C09140=1110.762,112.427,-59.197,-179.708,8.252,149.498
C09141=1110.767,112.179,-59.177,-179.709,8.249,149.498
C09142=1110.771,111.930,-59.156,-179.711,8.245,149.498
C09143=1110.776,111.680,-59.137,-179.713,8.242,149.498
C09144=1110.780,111.431,-59.116,-179.714,8.238,149.497
C09145=1110.786,111.182,-59.096,-179.716,8.235,149.497
C09146=1110.791,110.932,-59.077,-179.718,8.231,149.497
C09147=1110.795,110.683,-59.056,-179.720,8.228,149.496
C09148=1110.800,110.434,-59.037,-179.721,8.224,149.496
C09149=1110.805,110.185,-59.016,-179.724,8.221,149.496
C09150=1110.810,109.936,-58.997,-179.726,8.216,149.496
C09151=1110.814,109.687,-58.977,-179.728,8.213,149.495
C09152=1110.819,109.437,-58.957,-179.730,8.209,149.495
C09153=1110.824,109.188,-58.937,-179.732,8.205,149.495
C09154=1110.829,108.940,-58.917,-179.734,8.202,149.494
C09155=1110.834,108.690,-58.898,-179.736,8.198,149.494
C09156=1110.838,108.440,-58.878,-179.738,8.195,149.494
C09157=1110.843,108.192,-58.858,-179.740,8.191,149.494
C09158=1110.848,107.942,-58.838,-179.741,8.187,149.493
C09159=1110.852,107.693,-58.819,-179.743,8.184,149.493
C09160=1110.857,107.444,-58.799,-179.745,8.180,149.493
C09161=1110.861,107.195,-58.779,-179.747,8.176,149.492
C09162=1110.867,106.946,-58.760,-179.749,8.173,149.492
C09163=1110.871,106.697,-58.740,-179.751,8.169,149.492
C09164=1110.876,106.448,-58.720,-179.753,8.165,149.491
C09165=1110.881,106.198,-58.700,-179.754,8.161,149.491
C09166=1110.886,105.949,-58.681,-179.756,8.158,149.491
C09167=1110.890,105.736,-58.664,-179.758,8.154,149.490
C09168=1110.894,105.522,-58.647,-179.759,8.151,149.490
C09169=1110.898,105.308,-58.631,-179.761,8.149,149.490
C09170=1110.902,105.094,-58.613,-179.763,8.145,149.490
C09171=1110.906,104.880,-58.597,-179.764,8.142,149.489
C09172=1110.910,104.666,-58.580,-179.766,8.139,149.489
C09173=1110.914,104.453,-58.563,-179.767,8.135,149.488
C09174=1110.919,104.239,-58.547,-179.769,8.132,149.488
C09175=1110.923,103.989,-58.527,-179.771,8.128,149.488
C09176=1110.928,103.740,-58.507,-179.773,8.125,149.488
C09177=1110.932,103.492,-58.488,-179.774,8.121,149.487
C09178=1110.937,103.242,-58.468,-179.776,8.118,149.487
C09179=1110.942,102.993,-58.448,-179.777,8.114,149.487
C09180=1110.947,102.744,-58.429,-179.779,8.110,149.486
C09181=1110.952,102.494,-58.410,-179.781,8.106,149.486
C09182=1110.957,102.246,-58.391,-179.783,8.103,149.485
C09183=1110.961,101.996,-58.371,-179.784,8.099,149.485
C09184=1110.966,101.747,-58.352,-179.786,8.095,149.485
C09185=1110.971,101.498,-58.332,-179.787,8.091,149.484
C09186=1110.975,101.248,-58.313,-179.789,8.088,149.484
C09187=1110.980,100.999,-58.294,-179.791,8.084,149.483
C09188=1110.985,100.750,-58.274,-179.793,8.080,149.483
C09189=1110.990,100.500,-58.255,-179.794,8.076,149.483
C09190=1110.995,100.252,-58.236,-179.796,8.072,149.482
C09191=1111.000,100.002,-58.216,-179.798,8.069,149.482
C09192=1111.005,99.753,-58.197,-179.800,8.065,149.481
C09193=1111.009,99.504,-58.178,-179.801,8.061,149.481
C09194=1111.014,99.255,-58.158,-179.803,8.057,149.481
C09195=1111.019,99.006,-58.139,-179.804,8.053,149.480
C09196=1111.023,98.756,-58.120,-179.805,8.050,149.480
C09197=1111.029,98.507,-58.101,-179.807,8.046,149.479
C09198=1111.033,98.257,-58.082,-179.808,8.042,149.479
C09199=1111.038,98.009,-58.063,-179.811,8.039,149.479
C09200=1111.043,97.759,-58.043,-179.812,8.035,149.478
C09201=1111.047,97.511,-58.025,-179.814,8.031,149.478
C09202=1111.052,97.261,-58.005,-179.815,8.027,149.477
C09203=1111.058,97.012,-57.986,-179.817,8.023,149.477
C09204=1111.062,96.762,-57.967,-179.819,8.019,149.476
C09205=1111.067,96.514,-57.948,-179.820,8.015,149.476
C09206=1111.071,96.264,-57.929,-179.821,8.012,149.476
C09207=1111.076,96.015,-57.910,-179.823,8.008,149.475
C09208=1111.081,95.765,-57.891,-179.824,8.004,149.475
C09209=1111.086,95.517,-57.872,-179.826,8.001,149.474
C09210=1111.091,95.267,-57.852,-179.827,7.996,149.474
C09211=1111.095,95.019,-57.834,-179.829,7.992,149.473
C09212=1111.100,94.768,-57.815,-179.830,7.988,149.473
C09213=1111.105,94.520,-57.796,-179.831,7.985,149.472
C09214=1111.110,94.270,-57.776,-179.833,7.981,149.472
C09215=1111.115,94.021,-57.758,-179.834,7.978,149.471
C09216=1111.119,93.771,-57.739,-179.836,7.974,149.471
C09217=1111.124,93.523,-57.720,-179.838,7.970,149.471
C09218=1111.129,93.273,-57.701,-179.839,7.966,149.470
C09219=1111.134,93.024,-57.682,-179.840,7.962,149.470
C09220=1111.138,92.775,-57.663,-179.841,7.959,149.469
C09221=1111.143,92.525,-57.645,-179.843,7.955,149.469
C09222=1111.149,92.277,-57.625,-179.845,7.951,149.468
C09223=1111.153,92.062,-57.609,-179.846,7.948,149.468
C09224=1111.156,91.848,-57.593,-179.846,7.945,149.467
C09225=1111.161,91.635,-57.578,-179.847,7.941,149.467
C09226=1111.165,91.421,-57.561,-179.849,7.938,149.467
C09227=1111.169,91.206,-57.545,-179.850,7.934,149.466
C09228=1111.174,90.993,-57.529,-179.851,7.932,149.466
C09229=1111.177,90.779,-57.513,-179.852,7.929,149.465
C09230=1111.181,90.565,-57.497,-179.854,7.925,149.465
C09231=1111.187,90.316,-57.478,-179.855,7.921,149.464
C09232=1111.191,90.066,-57.459,-179.856,7.917,149.464
C09233=1111.195,89.818,-57.440,-179.858,7.913,149.463
C09234=1111.201,89.568,-57.422,-179.859,7.910,149.463
C09235=1111.205,89.319,-57.403,-179.860,7.906,149.462
C09236=1111.211,89.069,-57.384,-179.861,7.902,149.462
C09237=1111.215,88.821,-57.366,-179.863,7.898,149.462
C09238=1111.220,88.571,-57.347,-179.864,7.894,149.461
C09239=1111.225,88.322,-57.328,-179.865,7.891,149.460
C09240=1111.229,88.072,-57.310,-179.867,7.887,149.460
C09241=1111.234,87.824,-57.291,-179.868,7.883,149.459
C09242=1111.240,87.574,-57.272,-179.869,7.880,149.459
C09243=1111.244,87.325,-57.253,-179.870,7.876,149.459
C09244=1111.249,87.076,-57.235,-179.872,7.871,149.458
C09245=1111.254,86.826,-57.217,-179.873,7.868,149.457
C09246=1111.258,86.577,-57.198,-179.874,7.864,149.457
C09247=1111.263,86.328,-57.180,-179.875,7.860,149.456
C09248=1111.269,86.078,-57.161,-179.877,7.856,149.456
C09249=1111.273,85.829,-57.142,-179.877,7.853,149.455
C09250=1111.278,85.580,-57.124,-179.879,7.849,149.455
C09251=1111.283,85.331,-57.106,-179.880,7.846,149.454
C09252=1111.288,85.082,-57.087,-179.881,7.841,149.454
C09253=1111.292,84.832,-57.068,-179.883,7.838,149.453
C09254=1111.297,84.583,-57.050,-179.883,7.834,149.453
C09255=1111.302,84.334,-57.032,-179.885,7.830,149.452
C09256=1111.307,84.084,-57.013,-179.886,7.826,149.452
C09257=1111.312,83.835,-56.995,-179.887,7.823,149.451
C09258=1111.317,83.586,-56.977,-179.888,7.819,149.451
C09259=1111.321,83.337,-56.958,-179.889,7.815,149.450
C09260=1111.326,83.087,-56.940,-179.890,7.812,149.450
C09261=1111.331,82.838,-56.921,-179.892,7.807,149.449
C09262=1111.336,82.589,-56.903,-179.893,7.804,149.449
C09263=1111.341,82.340,-56.885,-179.894,7.800,149.448
C09264=1111.345,82.090,-56.866,-179.895,7.797,149.447
C09265=1111.350,81.841,-56.848,-179.896,7.792,149.447
C09266=1111.356,81.592,-56.830,-179.897,7.789,149.446
C09267=1111.361,81.342,-56.812,-179.898,7.785,149.446
C09268=1111.365,81.092,-56.793,-179.899,7.781,149.445
C09269=1111.369,80.844,-56.775,-179.900,7.778,149.445
C09270=1111.374,80.595,-56.757,-179.902,7.774,149.444
C09271=1111.379,80.346,-56.739,-179.902,7.770,149.444
C09272=1111.384,80.096,-56.721,-179.904,7.766,149.443
C09273=1111.389,79.846,-56.702,-179.904,7.763,149.443
C09274=1111.394,79.597,-56.684,-179.905,7.759,149.442
C09275=1111.399,79.348,-56.666,-179.906,7.756,149.441
C09276=1111.404,79.099,-56.648,-179.907,7.751,149.441
C09277=1111.409,78.849,-56.630,-179.908,7.748,149.440
C09278=1111.413,78.600,-56.611,-179.909,7.744,149.440
C09279=1111.418,78.386,-56.596,-179.910,7.741,149.439
C09280=1111.421,78.172,-56.580,-179.911,7.738,149.439
C09281=1111.426,77.958,-56.565,-179.912,7.734,149.438
C09282=1111.430,77.744,-56.549,-179.913,7.731,149.438
C09283=1111.435,77.530,-56.534,-179.914,7.728,149.437
C09284=1111.438,77.316,-56.518,-179.915,7.725,149.437
C09285=1111.442,77.103,-56.502,-179.916,7.722,149.436
C09286=1111.446,76.888,-56.487,-179.917,7.719,149.436
C09287=1111.451,76.639,-56.469,-179.917,7.715,149.435
C09288=1111.456,76.390,-56.451,-179.919,7.711,149.435
C09289=1111.461,76.141,-56.433,-179.920,7.707,149.435
C09290=1111.466,75.891,-56.415,-179.922,7.703,149.434
C09291=1111.471,75.642,-56.397,-179.923,7.699,149.433
C09292=1111.475,75.392,-56.379,-179.925,7.695,149.433
C09293=1111.480,75.143,-56.361,-179.926,7.691,149.433
C09294=1111.485,74.894,-56.343,-179.927,7.687,149.432
C09295=1111.490,74.645,-56.325,-179.929,7.683,149.431
C09296=1111.495,74.395,-56.307,-179.930,7.679,149.431
C09297=1111.500,74.146,-56.289,-179.932,7.675,149.431
C09298=1111.505,73.897,-56.272,-179.933,7.671,149.430
C09299=1111.510,73.647,-56.254,-179.935,7.667,149.430
C09300=1111.515,73.398,-56.236,-179.936,7.664,149.429
C09301=1111.520,73.149,-56.218,-179.937,7.660,149.428
C09302=1111.524,72.899,-56.199,-179.938,7.656,149.428
C09303=1111.529,72.649,-56.182,-179.940,7.652,149.428
C09304=1111.534,72.400,-56.164,-179.942,7.648,149.427
C09305=1111.539,72.151,-56.146,-179.943,7.644,149.426
C09306=1111.544,71.902,-56.128,-179.944,7.640,149.426
C09307=1111.548,71.653,-56.111,-179.946,7.636,149.426
C09308=1111.553,71.403,-56.093,-179.947,7.632,149.425
C09309=1111.558,71.154,-56.075,-179.948,7.628,149.425
C09310=1111.563,70.905,-56.057,-179.949,7.625,149.424
C09311=1111.568,70.656,-56.039,-179.951,7.620,149.423
C09312=1111.573,70.406,-56.022,-179.952,7.616,149.423
C09313=1111.578,70.157,-56.004,-179.954,7.612,149.423
C09314=1111.582,69.908,-55.987,-179.955,7.608,149.422
C09315=1111.588,69.658,-55.970,-179.956,7.604,149.422
C09316=1111.593,69.409,-55.952,-179.958,7.600,149.421
C09317=1111.597,69.160,-55.934,-179.959,7.596,149.420
C09318=1111.603,68.910,-55.916,-179.961,7.592,149.420
C09319=1111.608,68.661,-55.898,-179.962,7.588,149.420
C09320=1111.612,68.412,-55.881,-179.963,7.585,149.419
C09321=1111.617,68.162,-55.864,-179.964,7.581,149.418
C09322=1111.622,67.913,-55.846,-179.966,7.577,149.418
C09323=1111.627,67.664,-55.828,-179.967,7.573,149.417
C09324=1111.631,67.414,-55.811,-179.969,7.569,149.417
C09325=1111.636,67.165,-55.793,-179.970,7.565,149.417
C09326=1111.641,66.915,-55.776,-179.971,7.561,149.416
C09327=1111.646,66.666,-55.758,-179.973,7.557,149.415
C09328=1111.651,66.417,-55.741,-179.973,7.553,149.415
C09329=1111.656,66.167,-55.723,-179.975,7.549,149.414
C09330=1111.661,65.918,-55.706,-179.976,7.545,149.414
C09331=1111.666,65.669,-55.688,-179.978,7.541,149.413
C09332=1111.670,65.420,-55.671,-179.979,7.537,149.413
C09333=1111.675,65.170,-55.653,-179.981,7.533,149.412
C09334=1111.680,64.921,-55.635,-179.982,7.529,149.412
C09335=1111.684,64.707,-55.621,-179.983,7.526,149.411
C09336=1111.689,64.493,-55.606,-179.984,7.523,149.411
C09337=1111.692,64.279,-55.591,-179.985,7.519,149.410
C09338=1111.697,64.065,-55.576,-179.986,7.516,149.410
C09339=1111.701,63.851,-55.562,-179.987,7.513,149.410
C09340=1111.706,63.637,-55.547,-179.989,7.509,149.409
C09341=1111.710,63.422,-55.531,-179.990,7.506,149.409
C09342=1111.714,63.208,-55.517,-179.991,7.502,149.408
C09343=1111.719,62.959,-55.500,-179.992,7.498,149.408
C09344=1111.723,62.710,-55.482,-179.993,7.494,149.407
C09345=1111.728,62.460,-55.465,-179.994,7.490,149.407
C09346=1111.734,62.210,-55.448,-179.996,7.486,149.406
C09347=1111.738,61.961,-55.430,-179.997,7.483,149.406
C09348=1111.744,61.712,-55.413,-179.998,7.479,149.405
C09349=1111.748,61.463,-55.397,-179.999,7.475,149.405
C09350=1111.753,61.214,-55.379,179.999,7.470,149.404
C09351=1111.757,60.964,-55.362,179.998,7.467,149.404
C09352=1111.763,60.714,-55.345,179.997,7.462,149.403
C09353=1111.768,60.465,-55.327,179.995,7.458,149.402
C09354=1111.773,60.216,-55.310,179.995,7.455,149.402
C09355=1111.778,59.967,-55.293,179.993,7.451,149.401
C09356=1111.782,59.718,-55.276,179.992,7.447,149.401
C09357=1111.787,59.468,-55.259,179.990,7.443,149.400
C09358=1111.792,59.218,-55.242,179.989,7.439,149.400
C09359=1111.797,58.969,-55.225,179.988,7.435,149.399
C09360=1111.802,58.720,-55.208,179.987,7.431,149.399
C09361=1111.807,58.471,-55.190,179.986,7.427,149.398
C09362=1111.811,58.221,-55.174,179.984,7.423,149.398
C09363=1111.817,57.971,-55.156,179.983,7.419,149.397
C09364=1111.821,57.722,-55.140,179.982,7.415,149.397
C09365=1111.827,57.473,-55.123,179.980,7.411,149.396
C09366=1111.831,57.224,-55.105,179.979,7.407,149.396
C09367=1111.836,56.974,-55.088,179.978,7.403,149.395
C09368=1111.841,56.725,-55.072,179.977,7.399,149.394
C09369=1111.847,56.476,-55.055,179.976,7.395,149.394
C09370=1111.851,56.226,-55.038,179.974,7.391,149.393
C09371=1111.856,55.976,-55.021,179.973,7.387,149.393
C09372=1111.861,55.727,-55.004,179.972,7.383,149.392
C09373=1111.866,55.478,-54.988,179.971,7.379,149.392
C09374=1111.871,55.229,-54.970,179.970,7.375,149.391
C09375=1111.875,54.979,-54.953,179.968,7.371,149.391
C09376=1111.881,54.730,-54.936,179.967,7.367,149.390
C09377=1111.886,54.481,-54.920,179.966,7.363,149.389
C09378=1111.890,54.231,-54.903,179.965,7.359,149.389
C09379=1111.895,53.981,-54.886,179.964,7.356,149.388
C09380=1111.900,53.733,-54.869,179.963,7.351,149.388
C09381=1111.906,53.483,-54.852,179.962,7.347,149.387
C09382=1111.910,53.233,-54.835,179.960,7.343,149.387
C09383=1111.915,52.984,-54.819,179.959,7.339,149.386
C09384=1111.920,52.735,-54.802,179.958,7.336,149.386
C09385=1111.925,52.485,-54.785,179.957,7.331,149.385
C09386=1111.929,52.236,-54.768,179.956,7.327,149.384
C09387=1111.935,51.987,-54.752,179.954,7.323,149.384
C09388=1111.940,51.737,-54.735,179.953,7.319,149.383
C09389=1111.944,51.487,-54.719,179.952,7.315,149.383
C09390=1111.950,51.238,-54.702,179.951,7.311,149.382
C09391=1111.954,51.024,-54.688,179.950,7.308,149.382
C09392=1111.959,50.810,-54.674,179.949,7.304,149.381
C09393=1111.962,50.596,-54.659,179.948,7.301,149.381
C09394=1111.967,50.382,-54.644,179.947,7.297,149.380
C09395=1111.971,50.167,-54.630,179.946,7.294,149.380
C09396=1111.975,49.954,-54.616,179.945,7.290,149.379
C09397=1111.979,49.739,-54.602,179.944,7.287,149.379
C09398=1111.983,49.526,-54.588,179.943,7.283,149.378
C09399=1111.989,49.275,-54.571,179.942,7.280,149.378
C09400=1111.993,49.026,-54.555,179.941,7.276,149.377
C09401=1111.998,48.777,-54.538,179.940,7.272,149.376
C09402=1112.003,48.527,-54.522,179.939,7.267,149.376
C09403=1112.009,48.278,-54.505,179.937,7.263,149.375
C09404=1112.013,48.028,-54.489,179.936,7.259,149.375
C09405=1112.018,47.779,-54.472,179.936,7.256,149.374
C09406=1112.023,47.530,-54.456,179.934,7.251,149.373
C09407=1112.027,47.280,-54.439,179.933,7.247,149.373
C09408=1112.034,47.031,-54.423,179.932,7.243,149.372
C09409=1112.038,46.781,-54.406,179.931,7.239,149.372
C09410=1112.043,46.532,-54.390,179.930,7.236,149.371
C09411=1112.048,46.283,-54.373,179.929,7.231,149.371
C09412=1112.052,46.033,-54.357,179.928,7.227,149.370
C09413=1112.057,45.784,-54.341,179.927,7.223,149.369
C09414=1112.062,45.535,-54.324,179.925,7.219,149.369
C09415=1112.068,45.285,-54.308,179.925,7.215,149.368
C09416=1112.073,45.035,-54.292,179.923,7.211,149.368
C09417=1112.078,44.787,-54.275,179.922,7.207,149.367
C09418=1112.082,44.537,-54.259,179.921,7.203,149.366
C09419=1112.087,44.287,-54.243,179.920,7.198,149.366
C09420=1112.092,44.038,-54.226,179.919,7.194,149.365
C09421=1112.097,43.788,-54.210,179.918,7.191,149.364
C09422=1112.102,43.539,-54.194,179.917,7.187,149.364
C09423=1112.107,43.289,-54.178,179.916,7.182,149.363
C09424=1112.112,43.040,-54.162,179.915,7.178,149.363
C09425=1112.117,42.791,-54.145,179.913,7.174,149.362
C09426=1112.122,42.541,-54.129,179.913,7.170,149.361
C09427=1112.127,42.292,-54.112,179.911,7.166,149.361
C09428=1112.132,42.042,-54.097,179.910,7.162,149.360
C09429=1112.137,41.793,-54.080,179.909,7.158,149.360
C09430=1112.142,41.544,-54.064,179.908,7.154,149.359
C09431=1112.147,41.294,-54.048,179.908,7.150,149.358
C09432=1112.152,41.045,-54.032,179.907,7.146,149.358
C09433=1112.156,40.795,-54.015,179.905,7.142,149.357
C09434=1112.162,40.546,-54.000,179.904,7.137,149.357
C09435=1112.167,40.297,-53.984,179.903,7.133,149.356
C09436=1112.172,40.047,-53.968,179.903,7.130,149.355
C09437=1112.177,39.798,-53.951,179.901,7.125,149.355
C09438=1112.182,39.548,-53.935,179.900,7.121,149.354
C09439=1112.187,39.299,-53.920,179.899,7.117,149.353
C09440=1112.191,39.049,-53.903,179.898,7.112,149.353
C09441=1112.197,38.800,-53.888,179.897,7.108,149.352
C09442=1112.201,38.550,-53.871,179.896,7.105,149.352
C09443=1112.207,38.301,-53.855,179.895,7.101,149.351
C09444=1112.211,38.052,-53.840,179.894,7.096,149.350
C09445=1112.216,37.802,-53.824,179.893,7.092,149.350
C09446=1112.221,37.553,-53.808,179.892,7.088,149.349
C09447=1112.225,37.338,-53.794,179.892,7.084,149.348
C09448=1112.230,37.124,-53.781,179.891,7.081,149.348
C09449=1112.234,36.910,-53.767,179.890,7.078,149.347
C09450=1112.238,36.696,-53.753,179.889,7.074,149.347
C09451=1112.243,36.481,-53.740,179.888,7.070,149.346
C09452=1112.247,36.267,-53.726,179.887,7.067,149.346
C09453=1112.251,36.053,-53.712,179.887,7.064,149.345
C09454=1112.256,35.838,-53.698,179.886,7.059,149.344
C09455=1112.261,35.589,-53.682,179.885,7.055,149.344
C09456=1112.266,35.340,-53.666,179.884,7.051,149.343
C09457=1112.270,35.090,-53.651,179.883,7.047,149.342
C09458=1112.275,34.841,-53.636,179.882,7.043,149.342
C09459=1112.280,34.591,-53.619,179.881,7.038,149.341
C09460=1112.285,34.342,-53.603,179.880,7.034,149.341
C09461=1112.291,34.093,-53.588,179.880,7.031,149.340
C09462=1112.295,33.842,-53.572,179.878,7.026,149.339
C09463=1112.300,33.594,-53.556,179.877,7.022,149.339
C09464=1112.305,33.345,-53.540,179.876,7.018,149.338
C09465=1112.310,33.094,-53.524,179.875,7.013,149.337
C09466=1112.315,32.845,-53.509,179.875,7.010,149.337
C09467=1112.321,32.596,-53.493,179.874,7.006,149.336
C09468=1112.325,32.346,-53.478,179.873,7.001,149.335
C09469=1112.330,32.097,-53.462,179.872,6.997,149.335
C09470=1112.335,31.848,-53.446,179.871,6.993,149.334
C09471=1112.341,31.598,-53.430,179.870,6.989,149.333
C09472=1112.345,31.348,-53.415,179.869,6.985,149.333
C09473=1112.350,31.099,-53.400,179.868,6.980,149.332
C09474=1112.355,30.850,-53.384,179.867,6.976,149.331
C09475=1112.360,30.600,-53.368,179.866,6.971,149.330
C09476=1112.365,30.350,-53.353,179.865,6.967,149.330
C09477=1112.370,30.101,-53.337,179.865,6.964,149.329
C09478=1112.376,29.852,-53.322,179.864,6.959,149.329
C09479=1112.379,29.603,-53.306,179.863,6.955,149.328
C09480=1112.385,29.353,-53.290,179.862,6.951,149.327
C09481=1112.390,29.104,-53.275,179.861,6.946,149.326
C09482=1112.394,28.854,-53.259,179.861,6.942,149.326
C09483=1112.400,28.605,-53.244,179.860,6.938,149.325
C09484=1112.405,28.355,-53.228,179.859,6.934,149.324
C09485=1112.410,28.106,-53.213,179.858,6.930,149.324
C09486=1112.415,27.857,-53.197,179.857,6.925,149.323
C09487=1112.420,27.607,-53.182,179.856,6.921,149.322
C09488=1112.424,27.357,-53.167,179.855,6.917,149.322
C09489=1112.430,27.107,-53.152,179.854,6.913,149.321
C09490=1112.436,26.858,-53.136,179.854,6.908,149.320
C09491=1112.440,26.608,-53.121,179.853,6.904,149.319
C09492=1112.445,26.359,-53.105,179.852,6.899,149.319
C09493=1112.450,26.110,-53.090,179.851,6.896,149.318
C09494=1112.455,25.860,-53.075,179.851,6.891,149.317
C09495=1112.460,25.611,-53.059,179.850,6.887,149.316
C09496=1112.464,25.361,-53.044,179.849,6.883,149.316
C09497=1112.470,25.112,-53.028,179.848,6.878,149.315
C09498=1112.475,24.863,-53.013,179.847,6.874,149.314
C09499=1112.480,24.613,-52.998,179.847,6.870,149.314
C09500=1112.486,24.363,-52.983,179.845,6.866,149.313
C09501=1112.490,24.114,-52.968,179.845,6.861,149.312
C09502=1112.495,23.864,-52.952,179.844,6.857,149.311
C09503=1112.499,23.650,-52.940,179.843,6.853,149.311
C09504=1112.504,23.436,-52.926,179.843,6.850,149.310
C09505=1112.508,23.221,-52.912,179.842,6.845,149.309
C09506=1112.512,23.007,-52.900,179.842,6.842,149.309
C09507=1112.516,22.792,-52.886,179.841,6.839,149.308
C09508=1112.521,22.579,-52.874,179.840,6.834,149.308
C09509=1112.525,22.364,-52.860,179.839,6.831,149.307
C09510=1112.530,22.149,-52.847,179.839,6.827,149.306
C09511=1112.534,21.900,-52.832,179.838,6.823,149.306
C09512=1112.540,21.651,-52.817,179.837,6.818,149.305
C09513=1112.545,21.401,-52.802,179.836,6.814,149.304
C09514=1112.550,21.152,-52.787,179.836,6.810,149.303
C09515=1112.555,20.903,-52.772,179.835,6.806,149.303
C09516=1112.559,20.652,-52.756,179.834,6.801,149.302
C09517=1112.564,20.403,-52.742,179.833,6.797,149.301
C09518=1112.569,20.154,-52.727,179.833,6.792,149.300
C09519=1112.574,19.904,-52.711,179.832,6.788,149.300
C09520=1112.579,19.655,-52.697,179.831,6.783,149.299
C09521=1112.585,19.405,-52.681,179.831,6.779,149.298
C09522=1112.589,19.156,-52.666,179.830,6.775,149.297
C09523=1112.595,18.906,-52.651,179.829,6.770,149.297
C09524=1112.600,18.657,-52.636,179.829,6.766,149.296
C09525=1112.605,18.407,-52.622,179.828,6.761,149.295
C09526=1112.610,18.158,-52.606,179.827,6.757,149.294
C09527=1112.615,17.909,-52.591,179.827,6.753,149.293
C09528=1112.620,17.659,-52.577,179.826,6.748,149.293
C09529=1112.625,17.410,-52.562,179.825,6.744,149.292
C09530=1112.629,17.159,-52.547,179.824,6.739,149.291
C09531=1112.635,16.910,-52.531,179.823,6.735,149.290
C09532=1112.640,16.660,-52.517,179.823,6.730,149.290
C09533=1112.644,16.411,-52.502,179.822,6.726,149.289
C09534=1112.650,16.162,-52.487,179.822,6.722,149.288
C09535=1112.655,15.912,-52.472,179.821,6.717,149.287
C09536=1112.659,15.663,-52.457,179.820,6.713,149.286
C09537=1112.665,15.413,-52.442,179.820,6.708,149.286
C09538=1112.670,15.164,-52.427,179.819,6.704,149.285
C09539=1112.675,14.914,-52.413,179.818,6.699,149.284
C09540=1112.680,14.665,-52.398,179.818,6.695,149.283
C09541=1112.685,14.415,-52.383,179.818,6.691,149.282
C09542=1112.690,14.165,-52.369,179.817,6.686,149.282
C09543=1112.695,13.916,-52.354,179.816,6.682,149.281
C09544=1112.700,13.666,-52.339,179.815,6.677,149.280
C09545=1112.705,13.417,-52.324,179.814,6.673,149.279
C09546=1112.710,13.167,-52.310,179.814,6.668,149.278
C09547=1112.715,12.918,-52.295,179.813,6.663,149.277
C09548=1112.720,12.668,-52.280,179.813,6.660,149.277
C09549=1112.725,12.418,-52.266,179.812,6.655,149.276
C09550=1112.730,12.169,-52.251,179.812,6.650,149.275
C09551=1112.735,11.920,-52.237,179.811,6.646,149.274
C09552=1112.741,11.670,-52.222,179.810,6.641,149.273
C09553=1112.746,11.421,-52.207,179.810,6.637,149.273
C09554=1112.751,11.171,-52.193,179.809,6.632,149.272
C09555=1112.755,10.922,-52.178,179.809,6.627,149.271
C09556=1112.760,10.673,-52.163,179.809,6.623,149.270
C09557=1112.766,10.423,-52.149,179.808,6.619,149.269
C09558=1112.771,10.173,-52.134,179.807,6.614,149.268
C09559=1112.775,9.959,-52.121,179.806,6.610,149.268
C09560=1112.780,9.745,-52.108,179.806,6.606,149.267
C09561=1112.784,9.530,-52.096,179.806,6.603,149.266
C09562=1112.788,9.316,-52.084,179.805,6.598,149.265
C09563=1112.793,9.101,-52.071,179.805,6.594,149.265
C09564=1112.797,8.887,-52.059,179.804,6.591,149.264
C09565=1112.801,8.673,-52.047,179.803,6.586,149.263
C09566=1112.806,8.458,-52.034,179.803,6.582,149.262
C09567=1112.811,8.208,-52.019,179.803,6.578,149.261
C09568=1112.816,7.958,-52.005,179.802,6.573,149.261
C09569=1112.821,7.710,-51.990,179.801,6.569,149.260
C09570=1112.826,7.460,-51.976,179.801,6.564,149.259
C09571=1112.831,7.210,-51.962,179.800,6.559,149.258
C09572=1112.836,6.961,-51.948,179.800,6.555,149.257
C09573=1112.841,6.711,-51.933,179.800,6.551,149.256
C09574=1112.846,6.461,-51.919,179.799,6.546,149.256
C09575=1112.850,6.212,-51.904,179.798,6.542,149.255
C09576=1112.856,5.962,-51.889,179.798,6.537,149.254
C09577=1112.861,5.713,-51.875,179.797,6.532,149.253
C09578=1112.866,5.463,-51.861,179.796,6.528,149.252
C09579=1112.871,5.214,-51.847,179.795,6.523,149.252
C09580=1112.876,4.964,-51.832,179.795,6.518,149.251
C09581=1112.881,4.714,-51.818,179.794,6.514,149.250
C09582=1112.886,4.465,-51.804,179.794,6.509,149.249
C09583=1112.892,4.216,-51.790,179.793,6.505,149.248
C09584=1112.896,3.967,-51.775,179.792,6.500,149.247
C09585=1112.901,3.717,-51.761,179.792,6.496,149.246
C09586=1112.906,3.467,-51.746,179.792,6.491,149.246
C09587=1112.911,3.217,-51.732,179.791,6.487,149.245
C09588=1112.917,2.968,-51.718,179.790,6.482,149.244
C09589=1112.922,2.719,-51.704,179.790,6.478,149.243
C09590=1112.927,2.469,-51.690,179.789,6.473,149.242
C09591=1112.932,2.219,-51.675,179.789,6.468,149.241
C09592=1112.937,1.970,-51.662,179.788,6.464,149.241
C09593=1112.942,1.721,-51.647,179.787,6.459,149.240
C09594=1112.947,1.471,-51.633,179.787,6.454,149.239
C09595=1112.952,1.221,-51.619,179.787,6.451,149.238
C09596=1112.957,0.971,-51.604,179.786,6.446,149.237
C09597=1112.962,0.723,-51.591,179.785,6.441,149.236
C09598=1112.967,0.473,-51.577,179.785,6.437,149.236
C09599=1112.972,0.223,-51.563,179.784,6.432,149.235
C09600=1112.977,-0.027,-51.549,179.783,6.428,149.234
C09601=1112.983,-0.276,-51.535,179.783,6.423,149.233
C09602=1112.988,-0.526,-51.521,179.782,6.418,149.232
C09603=1112.993,-0.775,-51.507,179.781,6.414,149.232
C09604=1112.998,-1.024,-51.493,179.781,6.409,149.231
C09605=1113.003,-1.274,-51.478,179.781,6.405,149.230
C09606=1113.008,-1.524,-51.464,179.780,6.401,149.229
C09607=1113.012,-1.773,-51.450,179.779,6.396,149.228
C09608=1113.018,-2.023,-51.437,179.779,6.392,149.227
C09609=1113.023,-2.273,-51.423,179.778,6.387,149.226
C09610=1113.028,-2.522,-51.409,179.777,6.382,149.226
C09611=1113.034,-2.771,-51.395,179.777,6.378,149.225
C09612=1113.038,-3.021,-51.380,179.776,6.373,149.224
C09613=1113.044,-3.271,-51.367,179.775,6.369,149.223
C09614=1113.049,-3.520,-51.354,179.775,6.365,149.222
C09615=1113.052,-3.735,-51.341,179.774,6.360,149.222
C09616=1113.057,-3.949,-51.330,179.774,6.357,149.221
C09617=1113.061,-4.164,-51.317,179.773,6.352,149.220
C09618=1113.066,-4.378,-51.305,179.773,6.349,149.220
C09619=1113.070,-4.593,-51.293,179.772,6.345,149.219
C09620=1113.075,-4.807,-51.281,179.771,6.341,149.218
C09621=1113.080,-5.022,-51.270,179.771,6.337,149.218
C09622=1113.084,-5.237,-51.257,179.771,6.333,149.217
C09623=1113.088,-5.486,-51.244,179.770,6.329,149.216
C09624=1113.094,-5.736,-51.231,179.770,6.324,149.215
C09625=1113.099,-5.985,-51.216,179.769,6.320,149.214
C09626=1113.104,-6.234,-51.202,179.768,6.315,149.214
C09627=1113.109,-6.484,-51.189,179.768,6.310,149.213
C09628=1113.114,-6.734,-51.175,179.767,6.306,149.212
C09629=1113.119,-6.983,-51.161,179.767,6.301,149.211
C09630=1113.124,-7.233,-51.148,179.766,6.298,149.210
C09631=1113.129,-7.483,-51.134,179.766,6.293,149.209
C09632=1113.134,-7.732,-51.121,179.765,6.288,149.208
C09633=1113.139,-7.982,-51.106,179.764,6.284,149.208
C09634=1113.144,-8.231,-51.093,179.764,6.279,149.207
C09635=1113.150,-8.481,-51.080,179.763,6.274,149.206
C09636=1113.155,-8.730,-51.066,179.763,6.270,149.205
C09637=1113.160,-8.980,-51.053,179.762,6.265,149.204
C09638=1113.165,-9.230,-51.038,179.761,6.261,149.204
C09639=1113.170,-9.479,-51.025,179.761,6.256,149.203
C09640=1113.175,-9.729,-51.012,179.760,6.252,149.202
C09641=1113.180,-9.978,-50.998,179.760,6.248,149.201
C09642=1113.185,-10.228,-50.984,179.759,6.243,149.200
C09643=1113.190,-10.478,-50.970,179.759,6.238,149.199
C09644=1113.196,-10.727,-50.957,179.758,6.234,149.199
C09645=1113.200,-10.977,-50.943,179.757,6.229,149.198
C09646=1113.206,-11.226,-50.930,179.757,6.224,149.197
C09647=1113.211,-11.476,-50.916,179.756,6.220,149.196
C09648=1113.216,-11.725,-50.903,179.755,6.215,149.195
C09649=1113.221,-11.975,-50.889,179.755,6.211,149.194
C09650=1113.227,-12.225,-50.876,179.754,6.206,149.194
C09651=1113.231,-12.474,-50.862,179.754,6.201,149.193
C09652=1113.237,-12.724,-50.849,179.753,6.198,149.192
C09653=1113.241,-12.973,-50.835,179.753,6.193,149.191
C09654=1113.247,-13.223,-50.822,179.752,6.188,149.190
C09655=1113.251,-13.473,-50.809,179.752,6.183,149.189
C09656=1113.257,-13.722,-50.795,179.751,6.179,149.189
C09657=1113.261,-13.972,-50.782,179.750,6.174,149.188
C09658=1113.267,-14.221,-50.768,179.750,6.170,149.187
C09659=1113.272,-14.471,-50.755,179.749,6.165,149.186
C09660=1113.277,-14.720,-50.742,179.749,6.160,149.185
C09661=1113.282,-14.970,-50.728,179.748,6.156,149.184
C09662=1113.287,-15.219,-50.715,179.747,6.151,149.183
C09663=1113.293,-15.470,-50.702,179.747,6.146,149.183
C09664=1113.297,-15.718,-50.689,179.746,6.142,149.182
C09665=1113.303,-15.969,-50.675,179.746,6.137,149.181
C09666=1113.308,-16.218,-50.662,179.745,6.133,149.180
C09667=1113.312,-16.468,-50.649,179.745,6.129,149.179
C09668=1113.318,-16.717,-50.635,179.745,6.124,149.178
C09669=1113.323,-16.966,-50.623,179.744,6.119,149.177
C09670=1113.328,-17.217,-50.609,179.744,6.114,149.177
C09671=1113.333,-17.431,-50.598,179.743,6.110,149.176
C09672=1113.337,-17.645,-50.587,179.742,6.107,149.175
C09673=1113.341,-17.860,-50.575,179.742,6.102,149.174
C09674=1113.346,-18.075,-50.564,179.741,6.098,149.174
C09675=1113.350,-18.289,-50.552,179.741,6.095,149.173
C09676=1113.354,-18.504,-50.542,179.741,6.090,149.172
C09677=1113.359,-18.719,-50.530,179.740,6.086,149.171
C09678=1113.363,-18.933,-50.519,179.739,6.082,149.171
C09679=1113.369,-19.183,-50.506,179.739,6.077,149.170
C09680=1113.374,-19.433,-50.492,179.738,6.073,149.169
C09681=1113.379,-19.682,-50.479,179.738,6.068,149.168
C09682=1113.383,-19.932,-50.466,179.737,6.063,149.167
C09683=1113.389,-20.181,-50.453,179.737,6.058,149.166
C09684=1113.394,-20.431,-50.440,179.736,6.054,149.165
C09685=1113.399,-20.681,-50.427,179.736,6.049,149.164
C09686=1113.404,-20.930,-50.414,179.735,6.044,149.164
C09687=1113.410,-21.180,-50.402,179.735,6.040,149.163
C09688=1113.415,-21.429,-50.387,179.734,6.035,149.162
C09689=1113.420,-21.679,-50.375,179.734,6.030,149.161
C09690=1113.425,-21.928,-50.362,179.733,6.026,149.160
C09691=1113.430,-22.178,-50.349,179.732,6.021,149.159
C09692=1113.435,-22.428,-50.336,179.732,6.016,149.158
C09693=1113.440,-22.677,-50.323,179.731,6.012,149.157
C09694=1113.446,-22.927,-50.310,179.731,6.007,149.157
C09695=1113.451,-23.177,-50.297,179.731,6.002,149.156
C09696=1113.456,-23.426,-50.285,179.730,5.997,149.155
C09697=1113.461,-23.676,-50.271,179.730,5.993,149.154
C09698=1113.466,-23.926,-50.258,179.729,5.988,149.153
C09699=1113.471,-24.175,-50.246,179.729,5.983,149.152
C09700=1113.476,-24.425,-50.233,179.729,5.978,149.151
C09701=1113.482,-24.675,-50.220,179.728,5.973,149.150
C09702=1113.487,-24.924,-50.207,179.728,5.969,149.149
C09703=1113.492,-25.173,-50.194,179.727,5.964,149.148
C09704=1113.496,-25.423,-50.181,179.727,5.959,149.147
C09705=1113.502,-25.673,-50.168,179.726,5.954,149.146
C09706=1113.507,-25.922,-50.156,179.726,5.950,149.146
C09707=1113.512,-26.172,-50.143,179.726,5.945,149.144
C09708=1113.517,-26.422,-50.130,179.727,5.941,149.143
C09709=1113.522,-26.671,-50.117,179.727,5.937,149.142
C09710=1113.528,-26.920,-50.104,179.728,5.933,149.141
C09711=1113.533,-27.171,-50.092,179.727,5.928,149.140
C09712=1113.538,-27.420,-50.079,179.728,5.924,149.139
C09713=1113.543,-27.670,-50.067,179.728,5.920,149.138
C09714=1113.548,-27.919,-50.054,179.728,5.916,149.137
C09715=1113.554,-28.169,-50.041,179.728,5.911,149.136
C09716=1113.559,-28.419,-50.028,179.728,5.907,149.135
C09717=1113.564,-28.668,-50.015,179.728,5.903,149.134
C09718=1113.569,-28.917,-50.003,179.729,5.898,149.133
C09719=1113.574,-29.168,-49.991,179.729,5.894,149.132
C09720=1113.579,-29.417,-49.978,179.728,5.889,149.131
C09721=1113.584,-29.667,-49.965,179.728,5.885,149.131
C09722=1113.590,-29.916,-49.952,179.728,5.881,149.130
C09723=1113.594,-30.166,-49.939,179.728,5.876,149.129
C09724=1113.600,-30.416,-49.927,179.729,5.872,149.128
C09725=1113.605,-30.666,-49.915,179.728,5.867,149.127
C09726=1113.610,-30.915,-49.902,179.728,5.863,149.126
C09727=1113.615,-31.129,-49.891,179.728,5.860,149.125
C09728=1113.619,-31.344,-49.880,179.728,5.856,149.124
C09729=1113.623,-31.560,-49.869,179.728,5.852,149.124
C09730=1113.627,-31.774,-49.858,179.728,5.848,149.123
C09731=1113.632,-31.988,-49.847,179.728,5.845,149.122
C09732=1113.636,-32.203,-49.837,179.727,5.841,149.121
C09733=1113.641,-32.418,-49.826,179.727,5.837,149.120
C09734=1113.646,-32.633,-49.816,179.726,5.833,149.120
C09735=1113.651,-32.882,-49.803,179.727,5.829,149.119
C09736=1113.656,-33.131,-49.791,179.726,5.824,149.118
C09737=1113.660,-33.381,-49.778,179.726,5.820,149.117
C09738=1113.666,-33.631,-49.766,179.725,5.815,149.116
C09739=1113.671,-33.880,-49.753,179.725,5.811,149.115
C09740=1113.676,-34.130,-49.741,179.724,5.807,149.114
C09741=1113.681,-34.380,-49.729,179.724,5.802,149.114
C09742=1113.687,-34.629,-49.716,179.723,5.797,149.113
C09743=1113.691,-34.879,-49.703,179.723,5.792,149.112
C09744=1113.697,-35.129,-49.691,179.723,5.788,149.111
C09745=1113.702,-35.379,-49.678,179.722,5.784,149.110
C09746=1113.708,-35.628,-49.665,179.722,5.779,149.109
C09747=1113.713,-35.878,-49.654,179.721,5.775,149.108
C09748=1113.718,-36.127,-49.641,179.721,5.770,149.107
C09749=1113.723,-36.377,-49.628,179.720,5.765,149.107
C09750=1113.729,-36.626,-49.616,179.720,5.761,149.106
C09751=1113.732,-36.876,-49.604,179.719,5.756,149.105
C09752=1113.738,-37.126,-49.592,179.719,5.751,149.104
C09753=1113.743,-37.375,-49.580,179.718,5.747,149.103
C09754=1113.748,-37.625,-49.568,179.717,5.742,149.102
C09755=1113.754,-37.875,-49.555,179.716,5.737,149.102
C09756=1113.759,-38.125,-49.543,179.716,5.732,149.101
C09757=1113.764,-38.374,-49.531,179.715,5.727,149.100
C09758=1113.769,-38.623,-49.518,179.714,5.723,149.099
C09759=1113.775,-38.873,-49.506,179.714,5.718,149.098
C09760=1113.780,-39.123,-49.494,179.713,5.713,149.097
C09761=1113.785,-39.372,-49.482,179.712,5.708,149.096
C09762=1113.791,-39.622,-49.470,179.711,5.703,149.096
C09763=1113.796,-39.872,-49.457,179.710,5.698,149.095
C09764=1113.801,-40.122,-49.445,179.710,5.693,149.094
C09765=1113.805,-40.371,-49.433,179.709,5.688,149.093
C09766=1113.810,-40.621,-49.421,179.709,5.683,149.092
C09767=1113.816,-40.871,-49.408,179.707,5.678,149.091
C09768=1113.821,-41.121,-49.397,179.707,5.673,149.090
C09769=1113.826,-41.370,-49.385,179.706,5.667,149.090
C09770=1113.832,-41.620,-49.372,179.705,5.663,149.089
C09771=1113.837,-41.870,-49.360,179.704,5.657,149.088
C09772=1113.841,-42.119,-49.348,179.703,5.652,149.087
C09773=1113.847,-42.369,-49.336,179.702,5.647,149.086
C09774=1113.852,-42.619,-49.324,179.701,5.642,149.085
C09775=1113.857,-42.868,-49.312,179.700,5.636,149.084
C09776=1113.863,-43.118,-49.300,179.700,5.631,149.083
C09777=1113.867,-43.367,-49.289,179.701,5.627,149.082
C09778=1113.873,-43.617,-49.276,179.700,5.622,149.081
C09779=1113.878,-43.867,-49.264,179.700,5.617,149.080
C09780=1113.883,-44.117,-49.252,179.701,5.612,149.079
C09781=1113.889,-44.366,-49.241,179.701,5.607,149.078
C09782=1113.894,-44.615,-49.229,179.701,5.603,149.077
C09783=1113.898,-44.830,-49.219,179.701,5.599,149.076
C09784=1113.903,-45.045,-49.208,179.701,5.595,149.075
C09785=1113.908,-45.260,-49.198,179.702,5.590,149.074
C09786=1113.912,-45.475,-49.188,179.702,5.586,149.073
C09787=1113.916,-45.689,-49.177,179.702,5.583,149.072
C09788=1113.920,-45.904,-49.167,179.702,5.579,149.071
C09789=1113.925,-46.119,-49.157,179.702,5.575,149.070
C09790=1113.930,-46.334,-49.147,179.703,5.571,149.069
C09791=1113.934,-46.583,-49.135,179.703,5.566,149.068
C09792=1113.940,-46.833,-49.123,179.703,5.562,149.067
C09793=1113.945,-47.083,-49.111,179.703,5.556,149.066
C09794=1113.950,-47.333,-49.099,179.703,5.551,149.065
C09795=1113.955,-47.582,-49.088,179.703,5.547,149.064
C09796=1113.961,-47.832,-49.076,179.703,5.542,149.063
C09797=1113.967,-48.081,-49.064,179.704,5.538,149.062
C09798=1113.971,-48.330,-49.052,179.704,5.533,149.061
C09799=1113.978,-48.674,-49.036,179.704,5.526,149.059
C09800=1113.985,-49.015,-49.020,179.704,5.520,149.058
C09801=1113.993,-49.358,-49.004,179.704,5.513,149.056
C09802=1114.000,-49.700,-48.988,179.704,5.507,149.055
C09803=1114.005,-49.950,-48.976,179.705,5.503,149.054
C09804=1114.010,-50.199,-48.965,179.705,5.498,149.053
C09805=1114.015,-50.449,-48.953,179.705,5.493,149.052
C09806=1114.020,-50.699,-48.942,179.705,5.489,149.050
C09807=1114.025,-50.949,-48.930,179.705,5.483,149.049
C09808=1114.031,-51.198,-48.918,179.705,5.478,149.048
C09809=1114.036,-51.448,-48.907,179.706,5.474,149.047
C09810=1114.041,-51.697,-48.894,179.706,5.469,149.046
C09811=1114.046,-51.947,-48.883,179.706,5.465,149.045
C09812=1114.051,-52.197,-48.871,179.706,5.460,149.044
C09813=1114.057,-52.447,-48.859,179.706,5.455,149.043
C09814=1114.061,-52.696,-48.848,179.707,5.451,149.042
C09815=1114.068,-52.945,-48.836,179.706,5.446,149.041
C09816=1114.072,-53.195,-48.825,179.707,5.442,149.040
C09817=1114.078,-53.445,-48.813,179.707,5.436,149.039
C09818=1114.082,-53.695,-48.802,179.707,5.432,149.038
C09819=1114.088,-53.945,-48.790,179.707,5.427,149.036
C09820=1114.093,-54.194,-48.778,179.707,5.422,149.035
C09821=1114.098,-54.443,-48.767,179.707,5.418,149.034
C09822=1114.104,-54.693,-48.755,179.708,5.413,149.033
C09823=1114.109,-54.943,-48.744,179.708,5.408,149.032
C09824=1114.114,-55.193,-48.732,179.708,5.404,149.031
C09825=1114.119,-55.443,-48.721,179.708,5.399,149.030
C09826=1114.125,-55.692,-48.710,179.708,5.394,149.029
C09827=1114.130,-55.942,-48.699,179.708,5.390,149.028
C09828=1114.135,-56.192,-48.687,179.708,5.385,149.027
C09829=1114.140,-56.442,-48.676,179.709,5.381,149.026
C09830=1114.145,-56.691,-48.664,179.709,5.376,149.025
C09831=1114.151,-56.940,-48.653,179.709,5.371,149.024
C09832=1114.156,-57.190,-48.641,179.709,5.367,149.023
C09833=1114.161,-57.440,-48.630,179.709,5.361,149.021
C09834=1114.166,-57.690,-48.618,179.709,5.356,149.020
C09835=1114.171,-57.939,-48.607,179.709,5.352,149.019
C09836=1114.176,-58.189,-48.596,179.710,5.347,149.018
C09837=1114.182,-58.439,-48.584,179.710,5.343,149.017
C09838=1114.187,-58.689,-48.573,179.710,5.338,149.016
C09839=1114.194,-59.026,-48.558,179.710,5.332,149.015
C09840=1114.201,-59.362,-48.542,179.710,5.325,149.013
C09841=1114.208,-59.700,-48.527,179.710,5.319,149.012
C09842=1114.215,-60.037,-48.512,179.710,5.312,149.010
C09843=1114.220,-60.287,-48.500,179.710,5.308,149.009
C09844=1114.225,-60.536,-48.489,179.710,5.303,149.009
C09845=1114.230,-60.785,-48.478,179.709,5.297,149.008
C09846=1114.236,-61.036,-48.467,179.708,5.293,149.007
C09847=1114.241,-61.286,-48.455,179.708,5.287,149.006
C09848=1114.247,-61.535,-48.444,179.707,5.282,149.005
C09849=1114.252,-61.784,-48.433,179.707,5.277,149.004
C09850=1114.257,-62.035,-48.422,179.707,5.272,149.003
C09851=1114.262,-62.285,-48.410,179.706,5.267,149.002
C09852=1114.267,-62.533,-48.399,179.706,5.262,149.001
C09853=1114.272,-62.784,-48.389,179.705,5.257,149.000
C09854=1114.278,-63.034,-48.377,179.704,5.251,148.999
C09855=1114.283,-63.283,-48.366,179.704,5.247,148.998
C09856=1114.288,-63.533,-48.355,179.704,5.242,148.997
C09857=1114.293,-63.783,-48.343,179.704,5.237,148.996
C09858=1114.299,-64.032,-48.333,179.703,5.231,148.995
C09859=1114.304,-64.282,-48.322,179.703,5.226,148.994
C09860=1114.308,-64.532,-48.311,179.702,5.221,148.993
C09861=1114.314,-64.781,-48.299,179.702,5.215,148.992
C09862=1114.319,-65.031,-48.289,179.702,5.211,148.991
C09863=1114.324,-65.281,-48.277,179.701,5.206,148.990
C09864=1114.330,-65.531,-48.266,179.701,5.200,148.989
C09865=1114.335,-65.780,-48.255,179.700,5.195,148.988
C09866=1114.340,-66.029,-48.244,179.700,5.190,148.987
C09867=1114.345,-66.279,-48.234,179.700,5.185,148.986
C09868=1114.351,-66.529,-48.222,179.700,5.179,148.985
C09869=1114.356,-66.779,-48.212,179.699,5.175,148.984
C09870=1114.361,-67.028,-48.200,179.699,5.169,148.982
C09871=1114.367,-67.278,-48.190,179.699,5.165,148.981
C09872=1114.371,-67.528,-48.179,179.698,5.159,148.980
C09873=1114.377,-67.778,-48.168,179.698,5.154,148.979
C09874=1114.382,-68.027,-48.157,179.698,5.149,148.978
C09875=1114.387,-68.277,-48.146,179.698,5.144,148.977
C09876=1114.393,-68.526,-48.135,179.697,5.138,148.976
C09877=1114.398,-68.777,-48.125,179.698,5.133,148.975
C09878=1114.404,-69.026,-48.113,179.697,5.128,148.974
C09879=1114.409,-69.276,-48.103,179.697,5.123,148.973
C09880=1114.413,-69.526,-48.091,179.697,5.117,148.972
C09881=1114.419,-69.775,-48.081,179.696,5.112,148.971
C09882=1114.424,-70.025,-48.070,179.697,5.107,148.970
C09883=1114.429,-70.274,-48.060,179.697,5.102,148.968
C09884=1114.434,-70.525,-48.049,179.696,5.097,148.968
C09885=1114.440,-70.774,-48.037,179.696,5.091,148.966
C09886=1114.445,-71.024,-48.027,179.696,5.086,148.965
C09887=1114.451,-71.274,-48.017,179.696,5.081,148.964
C09888=1114.456,-71.523,-48.005,179.696,5.076,148.963
C09889=1114.461,-71.773,-47.995,179.696,5.071,148.962
C09890=1114.466,-72.023,-47.985,179.696,5.066,148.961
C09891=1114.471,-72.237,-47.975,179.696,5.061,148.960
C09892=1114.475,-72.452,-47.966,179.695,5.056,148.959
C09893=1114.480,-72.668,-47.957,179.696,5.052,148.958
C09894=1114.485,-72.882,-47.947,179.695,5.048,148.957
C09895=1114.489,-73.097,-47.939,179.696,5.043,148.956
C09896=1114.493,-73.313,-47.929,179.696,5.039,148.955
C09897=1114.498,-73.527,-47.920,179.696,5.035,148.954
C09898=1114.502,-73.742,-47.911,179.695,5.030,148.953
C09899=1114.508,-73.992,-47.901,179.696,5.025,148.952
C09900=1114.513,-74.242,-47.890,179.696,5.020,148.951
C09901=1114.519,-74.492,-47.879,179.696,5.014,148.950
C09902=1114.524,-74.741,-47.868,179.695,5.009,148.948
C09903=1114.529,-74.991,-47.858,179.695,5.004,148.948
C09904=1114.534,-75.241,-47.847,179.695,4.999,148.946
C09905=1114.540,-75.491,-47.837,179.695,4.993,148.945
C09906=1114.545,-75.740,-47.826,179.696,4.988,148.944
C09907=1114.550,-75.990,-47.816,179.696,4.983,148.943
C09908=1114.556,-76.239,-47.805,179.696,4.978,148.942
C09909=1114.561,-76.490,-47.795,179.696,4.973,148.941
C09910=1114.566,-76.739,-47.785,179.696,4.968,148.939
C09911=1114.572,-76.989,-47.774,179.696,4.963,148.938
C09912=1114.577,-77.238,-47.763,179.696,4.957,148.937
C09913=1114.582,-77.488,-47.753,179.697,4.952,148.936
C09914=1114.587,-77.738,-47.743,179.697,4.947,148.935
C09915=1114.592,-77.987,-47.733,179.697,4.942,148.933
C09916=1114.598,-78.237,-47.723,179.697,4.937,148.932
C09917=1114.603,-78.487,-47.712,179.697,4.932,148.931
C09918=1114.608,-78.737,-47.702,179.697,4.927,148.930
C09919=1114.613,-78.987,-47.691,179.698,4.921,148.929
C09920=1114.619,-79.236,-47.680,179.698,4.916,148.928
C09921=1114.624,-79.485,-47.670,179.698,4.911,148.926
C09922=1114.629,-79.736,-47.659,179.698,4.906,148.925
C09923=1114.635,-79.985,-47.649,179.698,4.901,148.924
C09924=1114.640,-80.235,-47.639,179.698,4.896,148.923
C09925=1114.645,-80.485,-47.628,179.698,4.890,148.922
C09926=1114.651,-80.734,-47.618,179.699,4.885,148.921
C09927=1114.655,-80.984,-47.608,179.699,4.880,148.919
C09928=1114.661,-81.234,-47.598,179.699,4.875,148.918
C09929=1114.666,-81.483,-47.588,179.699,4.870,148.917
C09930=1114.671,-81.734,-47.577,179.699,4.865,148.916
C09931=1114.677,-81.983,-47.567,179.699,4.860,148.915
C09932=1114.683,-82.233,-47.557,179.700,4.854,148.914
C09933=1114.687,-82.483,-47.547,179.700,4.849,148.912
C09934=1114.692,-82.732,-47.537,179.700,4.844,148.911
C09935=1114.698,-82.982,-47.526,179.701,4.839,148.910
C09936=1114.703,-83.232,-47.516,179.701,4.834,148.909
C09937=1114.709,-83.482,-47.506,179.702,4.829,148.907
C09938=1114.714,-83.731,-47.495,179.702,4.824,148.906
C09939=1114.719,-83.981,-47.486,179.702,4.819,148.905
C09940=1114.724,-84.231,-47.475,179.702,4.814,148.904
C09941=1114.730,-84.480,-47.465,179.702,4.808,148.903
C09942=1114.736,-84.730,-47.456,179.703,4.804,148.902
C09943=1114.741,-84.981,-47.445,179.704,4.799,148.900
C09944=1114.746,-85.230,-47.435,179.704,4.793,148.899
C09945=1114.751,-85.479,-47.425,179.704,4.788,148.898
C09946=1114.756,-85.730,-47.415,179.704,4.783,148.897
C09947=1114.761,-85.944,-47.406,179.705,4.779,148.896
C09948=1114.765,-86.160,-47.397,179.705,4.775,148.894
C09949=1114.770,-86.374,-47.389,179.706,4.771,148.894
C09950=1114.774,-86.589,-47.380,179.706,4.766,148.892
C09951=1114.779,-86.805,-47.372,179.706,4.762,148.891
C09952=1114.783,-87.020,-47.363,179.707,4.757,148.890
C09953=1114.788,-87.235,-47.354,179.707,4.753,148.889
C09954=1114.792,-87.450,-47.345,179.707,4.749,148.888
C09955=1114.798,-87.699,-47.335,179.708,4.744,148.887
C09956=1114.803,-87.949,-47.326,179.708,4.739,148.886
C09957=1114.809,-88.199,-47.316,179.708,4.734,148.885
C09958=1114.814,-88.449,-47.306,179.709,4.729,148.883
C09959=1114.819,-88.698,-47.295,179.709,4.724,148.882
C09960=1114.824,-88.948,-47.286,179.710,4.719,148.881
C09961=1114.830,-89.197,-47.276,179.711,4.714,148.880
C09962=1114.836,-89.447,-47.266,179.711,4.709,148.878
C09963=1114.840,-89.697,-47.256,179.711,4.704,148.877
C09964=1114.845,-89.947,-47.246,179.712,4.700,148.876
C09965=1114.851,-90.196,-47.236,179.712,4.694,148.875
C09966=1114.856,-90.446,-47.227,179.712,4.689,148.874
C09967=1114.861,-90.697,-47.216,179.713,4.685,148.872
C09968=1114.867,-90.946,-47.206,179.714,4.679,148.871
C09969=1114.872,-91.195,-47.196,179.715,4.675,148.870
C09970=1114.878,-91.445,-47.187,179.715,4.670,148.869
C09971=1114.882,-91.695,-47.177,179.715,4.665,148.867
C09972=1114.887,-91.945,-47.167,179.716,4.660,148.866
C09973=1114.893,-92.195,-47.157,179.716,4.655,148.865
C09974=1114.898,-92.444,-47.148,179.717,4.651,148.864
C09975=1114.904,-92.694,-47.137,179.717,4.645,148.863
C09976=1114.909,-92.943,-47.127,179.718,4.641,148.861
C09977=1114.914,-93.194,-47.118,179.718,4.636,148.860
C09978=1114.920,-93.444,-47.108,179.719,4.632,148.859
C09979=1114.925,-93.693,-47.099,179.719,4.626,148.858
C09980=1114.930,-93.943,-47.089,179.720,4.622,148.857
C09981=1114.936,-94.192,-47.078,179.721,4.616,148.855
C09982=1114.941,-94.442,-47.069,179.722,4.612,148.854
C09983=1114.946,-94.693,-47.059,179.722,4.607,148.853
C09984=1114.951,-94.942,-47.049,179.722,4.602,148.852
C09985=1114.957,-95.192,-47.040,179.722,4.597,148.851
C09986=1114.962,-95.441,-47.030,179.723,4.593,148.849
C09987=1114.967,-95.691,-47.020,179.723,4.588,148.848
C09988=1114.973,-95.941,-47.010,179.723,4.582,148.847
C09989=1114.978,-96.190,-47.001,179.724,4.578,148.846
C09990=1114.983,-96.441,-46.991,179.724,4.573,148.845
C09991=1114.988,-96.690,-46.981,179.724,4.568,148.843
C09992=1114.994,-96.940,-46.972,179.724,4.563,148.842
C09993=1114.999,-97.190,-46.962,179.725,4.558,148.841
C09994=1115.005,-97.440,-46.953,179.725,4.553,148.840
C09995=1115.010,-97.689,-46.943,179.726,4.548,148.839
C09996=1115.015,-97.939,-46.933,179.726,4.543,148.838
//INST
///DATE 2021/06/25 14:33
///ATTR SC,RW,RJ
////FRAME ROBOT
///GROUP1 RB1
NOP
MOVL C00000 V=800.0 PL=0
MOVL C00001 V=800.0 PL=0
MOVL C00002 V=800.0 PL=0
MOVL C00003 V=800.0 PL=0
MOVL C00004 V=800.0 PL=0
MOVL C00005 V=800.0 PL=0
MOVL C00006 V=800.0 PL=0
MOVL C00007 V=800.0 PL=0
MOVL C00008 V=800.0 PL=0
MOVL C00009 V=800.0 PL=0
MOVL C00010 V=800.0 PL=0
MOVL C00011 V=800.0 PL=0
MOVL C00012 V=800.0 PL=0
MOVL C00013 V=800.0 PL=0
MOVL C00014 V=800.0 PL=0
MOVL C00015 V=800.0 PL=0
MOVL C00016 V=800.0 PL=0
MOVL C00017 V=800.0 PL=0
MOVL C00018 V=800.0 PL=0
MOVL C00019 V=800.0 PL=0
MOVL C00020 V=800.0 PL=0
MOVL C00021 V=800.0 PL=0
MOVL C00022 V=800.0 PL=0
MOVL C00023 V=800.0 PL=0
MOVL C00024 V=800.0 PL=0
MOVL C00025 V=800.0 PL=0
MOVL C00026 V=800.0 PL=0
MOVL C00027 V=800.0 PL=0
MOVL C00028 V=800.0 PL=0
MOVL C00029 V=800.0 PL=0
MOVL C00030 V=800.0 PL=0
MOVL C00031 V=800.0 PL=0
MOVL C00032 V=800.0 PL=0
MOVL C00033 V=800.0 PL=0
MOVL C00034 V=800.0 PL=0
MOVL C00035 V=800.0 PL=0
MOVL C00036 V=800.0 PL=0
MOVL C00037 V=800.0 PL=0
MOVL C00038 V=800.0 PL=0
MOVL C00039 V=800.0 PL=0
MOVL C00040 V=800.0 PL=0
MOVL C00041 V=800.0 PL=0
MOVL C00042 V=800.0 PL=0
MOVL C00043 V=800.0 PL=0
MOVL C00044 V=800.0 PL=0
MOVL C00045 V=800.0 PL=0
MOVL C00046 V=800.0 PL=0
MOVL C00047 V=800.0 PL=0
MOVL C00048 V=800.0 PL=0
MOVL C00049 V=800.0 PL=0
MOVL C00050 V=800.0 PL=0
MOVL C00051 V=800.0 PL=0
MOVL C00052 V=800.0 PL=0
MOVL C00053 V=800.0 PL=0
MOVL C00054 V=800.0 PL=0
MOVL C00055 V=800.0 PL=0
MOVL C00056 V=800.0 PL=0
MOVL C00057 V=800.0 PL=0
MOVL C00058 V=800.0 PL=0
MOVL C00059 V=800.0 PL=0
MOVL C00060 V=800.0 PL=0
MOVL C00061 V=800.0 PL=0
MOVL C00062 V=800.0 PL=0
MOVL C00063 V=800.0 PL=0
MOVL C00064 V=800.0 PL=0
MOVL C00065 V=800.0 PL=0
MOVL C00066 V=800.0 PL=0
MOVL C00067 V=800.0 PL=0
MOVL C00068 V=800.0 PL=0
MOVL C00069 V=800.0 PL=0
MOVL C00070 V=800.0 PL=0
MOVL C00071 V=800.0 PL=0
MOVL C00072 V=800.0 PL=0
MOVL C00073 V=800.0 PL=0
MOVL C00074 V=800.0 PL=0
MOVL C00075 V=800.0 PL=0
MOVL C00076 V=800.0 PL=0
MOVL C00077 V=800.0 PL=0
MOVL C00078 V=800.0 PL=0
MOVL C00079 V=800.0 PL=0
MOVL C00080 V=800.0 PL=0
MOVL C00081 V=800.0 PL=0
MOVL C00082 V=800.0 PL=0
MOVL C00083 V=800.0 PL=0
MOVL C00084 V=800.0 PL=0
MOVL C00085 V=800.0 PL=0
MOVL C00086 V=800.0 PL=0
MOVL C00087 V=800.0 PL=0
MOVL C00088 V=800.0 PL=0
MOVL C00089 V=800.0 PL=0
MOVL C00090 V=800.0 PL=0
MOVL C00091 V=800.0 PL=0
MOVL C00092 V=800.0 PL=0
MOVL C00093 V=800.0 PL=0
MOVL C00094 V=800.0 PL=0
MOVL C00095 V=800.0 PL=0
MOVL C00096 V=800.0 PL=0
MOVL C00097 V=800.0 PL=0
MOVL C00098 V=800.0 PL=0
MOVL C00099 V=800.0 PL=0
MOVL C00100 V=800.0 PL=0
MOVL C00101 V=800.0 PL=0
MOVL C00102 V=800.0 PL=0
MOVL C00103 V=800.0 PL=0
MOVL C00104 V=800.0 PL=0
MOVL C00105 V=800.0 PL=0
MOVL C00106 V=800.0 PL=0
MOVL C00107 V=800.0 PL=0
MOVL C00108 V=800.0 PL=0
MOVL C00109 V=800.0 PL=0
MOVL C00110 V=800.0 PL=0
MOVL C00111 V=800.0 PL=0
MOVL C00112 V=800.0 PL=0
MOVL C00113 V=800.0 PL=0
MOVL C00114 V=800.0 PL=0
MOVL C00115 V=800.0 PL=0
MOVL C00116 V=800.0 PL=0
MOVL C00117 V=800.0 PL=0
MOVL C00118 V=800.0 PL=0
MOVL C00119 V=800.0 PL=0
MOVL C00120 V=800.0 PL=0
MOVL C00121 V=800.0 PL=0
MOVL C00122 V=800.0 PL=0
MOVL C00123 V=800.0 PL=0
MOVL C00124 V=800.0 PL=0
MOVL C00125 V=800.0 PL=0
MOVL C00126 V=800.0 PL=0
MOVL C00127 V=800.0 PL=0
MOVL C00128 V=800.0 PL=0
MOVL C00129 V=800.0 PL=0
MOVL C00130 V=800.0 PL=0
MOVL C00131 V=800.0 PL=0
MOVL C00132 V=800.0 PL=0
MOVL C00133 V=800.0 PL=0
MOVL C00134 V=800.0 PL=0
MOVL C00135 V=800.0 PL=0
MOVL C00136 V=800.0 PL=0
MOVL C00137 V=800.0 PL=0
MOVL C00138 V=800.0 PL=0
MOVL C00139 V=800.0 PL=0
MOVL C00140 V=800.0 PL=0
MOVL C00141 V=800.0 PL=0
MOVL C00142 V=800.0 PL=0
MOVL C00143 V=800.0 PL=0
MOVL C00144 V=800.0 PL=0
MOVL C00145 V=800.0 PL=0
MOVL C00146 V=800.0 PL=0
MOVL C00147 V=800.0 PL=0
MOVL C00148 V=800.0 PL=0
MOVL C00149 V=800.0 PL=0
MOVL C00150 V=800.0 PL=0
MOVL C00151 V=800.0 PL=0
MOVL C00152 V=800.0 PL=0
MOVL C00153 V=800.0 PL=0
MOVL C00154 V=800.0 PL=0
MOVL C00155 V=800.0 PL=0
MOVL C00156 V=800.0 PL=0
MOVL C00157 V=800.0 PL=0
MOVL C00158 V=800.0 PL=0
MOVL C00159 V=800.0 PL=0
MOVL C00160 V=800.0 PL=0
MOVL C00161 V=800.0 PL=0
MOVL C00162 V=800.0 PL=0
MOVL C00163 V=800.0 PL=0
MOVL C00164 V=800.0 PL=0
MOVL C00165 V=800.0 PL=0
MOVL C00166 V=800.0 PL=0
MOVL C00167 V=800.0 PL=0
MOVL C00168 V=800.0 PL=0
MOVL C00169 V=800.0 PL=0
MOVL C00170 V=800.0 PL=0
MOVL C00171 V=800.0 PL=0
MOVL C00172 V=800.0 PL=0
MOVL C00173 V=800.0 PL=0
MOVL C00174 V=800.0 PL=0
MOVL C00175 V=800.0 PL=0
MOVL C00176 V=800.0 PL=0
MOVL C00177 V=800.0 PL=0
MOVL C00178 V=800.0 PL=0
MOVL C00179 V=800.0 PL=0
MOVL C00180 V=800.0 PL=0
MOVL C00181 V=800.0 PL=0
MOVL C00182 V=800.0 PL=0
MOVL C00183 V=800.0 PL=0
MOVL C00184 V=800.0 PL=0
MOVL C00185 V=800.0 PL=0
MOVL C00186 V=800.0 PL=0
MOVL C00187 V=800.0 PL=0
MOVL C00188 V=800.0 PL=0
MOVL C00189 V=800.0 PL=0
MOVL C00190 V=800.0 PL=0
MOVL C00191 V=800.0 PL=0
MOVL C00192 V=800.0 PL=0
MOVL C00193 V=800.0 PL=0
MOVL C00194 V=800.0 PL=0
MOVL C00195 V=800.0 PL=0
MOVL C00196 V=800.0 PL=0
MOVL C00197 V=800.0 PL=0
MOVL C00198 V=800.0 PL=0
MOVL C00199 V=800.0 PL=0
MOVL C00200 V=800.0 PL=0
MOVL C00201 V=800.0 PL=0
MOVL C00202 V=800.0 PL=0
MOVL C00203 V=800.0 PL=0
MOVL C00204 V=800.0 PL=0
MOVL C00205 V=800.0 PL=0
MOVL C00206 V=800.0 PL=0
MOVL C00207 V=800.0 PL=0
MOVL C00208 V=800.0 PL=0
MOVL C00209 V=800.0 PL=0
MOVL C00210 V=800.0 PL=0
MOVL C00211 V=800.0 PL=0
MOVL C00212 V=800.0 PL=0
MOVL C00213 V=800.0 PL=0
MOVL C00214 V=800.0 PL=0
MOVL C00215 V=800.0 PL=0
MOVL C00216 V=800.0 PL=0
MOVL C00217 V=800.0 PL=0
MOVL C00218 V=800.0 PL=0
MOVL C00219 V=800.0 PL=0
MOVL C00220 V=800.0 PL=0
MOVL C00221 V=800.0 PL=0
MOVL C00222 V=800.0 PL=0
MOVL C00223 V=800.0 PL=0
MOVL C00224 V=800.0 PL=0
MOVL C00225 V=800.0 PL=0
MOVL C00226 V=800.0 PL=0
MOVL C00227 V=800.0 PL=0
MOVL C00228 V=800.0 PL=0
MOVL C00229 V=800.0 PL=0
MOVL C00230 V=800.0 PL=0
MOVL C00231 V=800.0 PL=0
MOVL C00232 V=800.0 PL=0
MOVL C00233 V=800.0 PL=0
MOVL C00234 V=800.0 PL=0
MOVL C00235 V=800.0 PL=0
MOVL C00236 V=800.0 PL=0
MOVL C00237 V=800.0 PL=0
MOVL C00238 V=800.0 PL=0
MOVL C00239 V=800.0 PL=0
MOVL C00240 V=800.0 PL=0
MOVL C00241 V=800.0 PL=0
MOVL C00242 V=800.0 PL=0
MOVL C00243 V=800.0 PL=0
MOVL C00244 V=800.0 PL=0
MOVL C00245 V=800.0 PL=0
MOVL C00246 V=800.0 PL=0
MOVL C00247 V=800.0 PL=0
MOVL C00248 V=800.0 PL=0
MOVL C00249 V=800.0 PL=0
MOVL C00250 V=800.0 PL=0
MOVL C00251 V=800.0 PL=0
MOVL C00252 V=800.0 PL=0
MOVL C00253 V=800.0 PL=0
MOVL C00254 V=800.0 PL=0
MOVL C00255 V=800.0 PL=0
MOVL C00256 V=800.0 PL=0
MOVL C00257 V=800.0 PL=0
MOVL C00258 V=800.0 PL=0
MOVL C00259 V=800.0 PL=0
MOVL C00260 V=800.0 PL=0
MOVL C00261 V=800.0 PL=0
MOVL C00262 V=800.0 PL=0
MOVL C00263 V=800.0 PL=0
MOVL C00264 V=800.0 PL=0
MOVL C00265 V=800.0 PL=0
MOVL C00266 V=800.0 PL=0
MOVL C00267 V=800.0 PL=0
MOVL C00268 V=800.0 PL=0
MOVL C00269 V=800.0 PL=0
MOVL C00270 V=800.0 PL=0
MOVL C00271 V=800.0 PL=0
MOVL C00272 V=800.0 PL=0
MOVL C00273 V=800.0 PL=0
MOVL C00274 V=800.0 PL=0
MOVL C00275 V=800.0 PL=0
MOVL C00276 V=800.0 PL=0
MOVL C00277 V=800.0 PL=0
MOVL C00278 V=800.0 PL=0
MOVL C00279 V=800.0 PL=0
MOVL C00280 V=800.0 PL=0
MOVL C00281 V=800.0 PL=0
MOVL C00282 V=800.0 PL=0
MOVL C00283 V=800.0 PL=0
MOVL C00284 V=800.0 PL=0
MOVL C00285 V=800.0 PL=0
MOVL C00286 V=800.0 PL=0
MOVL C00287 V=800.0 PL=0
MOVL C00288 V=800.0 PL=0
MOVL C00289 V=800.0 PL=0
MOVL C00290 V=800.0 PL=0
MOVL C00291 V=800.0 PL=0
MOVL C00292 V=800.0 PL=0
MOVL C00293 V=800.0 PL=0
MOVL C00294 V=800.0 PL=0
MOVL C00295 V=800.0 PL=0
MOVL C00296 V=800.0 PL=0
MOVL C00297 V=800.0 PL=0
MOVL C00298 V=800.0 PL=0
MOVL C00299 V=800.0 PL=0
MOVL C00300 V=800.0 PL=0
MOVL C00301 V=800.0 PL=0
MOVL C00302 V=800.0 PL=0
MOVL C00303 V=800.0 PL=0
MOVL C00304 V=800.0 PL=0
MOVL C00305 V=800.0 PL=0
MOVL C00306 V=800.0 PL=0
MOVL C00307 V=800.0 PL=0
MOVL C00308 V=800.0 PL=0
MOVL C00309 V=800.0 PL=0
MOVL C00310 V=800.0 PL=0
MOVL C00311 V=800.0 PL=0
MOVL C00312 V=800.0 PL=0
MOVL C00313 V=800.0 PL=0
MOVL C00314 V=800.0 PL=0
MOVL C00315 V=800.0 PL=0
MOVL C00316 V=800.0 PL=0
MOVL C00317 V=800.0 PL=0
MOVL C00318 V=800.0 PL=0
MOVL C00319 V=800.0 PL=0
MOVL C00320 V=800.0 PL=0
MOVL C00321 V=800.0 PL=0
MOVL C00322 V=800.0 PL=0
MOVL C00323 V=800.0 PL=0
MOVL C00324 V=800.0 PL=0
MOVL C00325 V=800.0 PL=0
MOVL C00326 V=800.0 PL=0
MOVL C00327 V=800.0 PL=0
MOVL C00328 V=800.0 PL=0
MOVL C00329 V=800.0 PL=0
MOVL C00330 V=800.0 PL=0
MOVL C00331 V=800.0 PL=0
MOVL C00332 V=800.0 PL=0
MOVL C00333 V=800.0 PL=0
MOVL C00334 V=800.0 PL=0
MOVL C00335 V=800.0 PL=0
MOVL C00336 V=800.0 PL=0
MOVL C00337 V=800.0 PL=0
MOVL C00338 V=800.0 PL=0
MOVL C00339 V=800.0 PL=0
MOVL C00340 V=800.0 PL=0
MOVL C00341 V=800.0 PL=0
MOVL C00342 V=800.0 PL=0
MOVL C00343 V=800.0 PL=0
MOVL C00344 V=800.0 PL=0
MOVL C00345 V=800.0 PL=0
MOVL C00346 V=800.0 PL=0
MOVL C00347 V=800.0 PL=0
MOVL C00348 V=800.0 PL=0
MOVL C00349 V=800.0 PL=0
MOVL C00350 V=800.0 PL=0
MOVL C00351 V=800.0 PL=0
MOVL C00352 V=800.0 PL=0
MOVL C00353 V=800.0 PL=0
MOVL C00354 V=800.0 PL=0
MOVL C00355 V=800.0 PL=0
MOVL C00356 V=800.0 PL=0
MOVL C00357 V=800.0 PL=0
MOVL C00358 V=800.0 PL=0
MOVL C00359 V=800.0 PL=0
MOVL C00360 V=800.0 PL=0
MOVL C00361 V=800.0 PL=0
MOVL C00362 V=800.0 PL=0
MOVL C00363 V=800.0 PL=0
MOVL C00364 V=800.0 PL=0
MOVL C00365 V=800.0 PL=0
MOVL C00366 V=800.0 PL=0
MOVL C00367 V=800.0 PL=0
MOVL C00368 V=800.0 PL=0
MOVL C00369 V=800.0 PL=0
MOVL C00370 V=800.0 PL=0
MOVL C00371 V=800.0 PL=0
MOVL C00372 V=800.0 PL=0
MOVL C00373 V=800.0 PL=0
MOVL C00374 V=800.0 PL=0
MOVL C00375 V=800.0 PL=0
MOVL C00376 V=800.0 PL=0
MOVL C00377 V=800.0 PL=0
MOVL C00378 V=800.0 PL=0
MOVL C00379 V=800.0 PL=0
MOVL C00380 V=800.0 PL=0
MOVL C00381 V=800.0 PL=0
MOVL C00382 V=800.0 PL=0
MOVL C00383 V=800.0 PL=0
MOVL C00384 V=800.0 PL=0
MOVL C00385 V=800.0 PL=0
MOVL C00386 V=800.0 PL=0
MOVL C00387 V=800.0 PL=0
MOVL C00388 V=800.0 PL=0
MOVL C00389 V=800.0 PL=0
MOVL C00390 V=800.0 PL=0
MOVL C00391 V=800.0 PL=0
MOVL C00392 V=800.0 PL=0
MOVL C00393 V=800.0 PL=0
MOVL C00394 V=800.0 PL=0
MOVL C00395 V=800.0 PL=0
MOVL C00396 V=800.0 PL=0
MOVL C00397 V=800.0 PL=0
MOVL C00398 V=800.0 PL=0
MOVL C00399 V=800.0 PL=0
MOVL C00400 V=800.0 PL=0
MOVL C00401 V=800.0 PL=0
MOVL C00402 V=800.0 PL=0
MOVL C00403 V=800.0 PL=0
MOVL C00404 V=800.0 PL=0
MOVL C00405 V=800.0 PL=0
MOVL C00406 V=800.0 PL=0
MOVL C00407 V=800.0 PL=0
MOVL C00408 V=800.0 PL=0
MOVL C00409 V=800.0 PL=0
MOVL C00410 V=800.0 PL=0
MOVL C00411 V=800.0 PL=0
MOVL C00412 V=800.0 PL=0
MOVL C00413 V=800.0 PL=0
MOVL C00414 V=800.0 PL=0
MOVL C00415 V=800.0 PL=0
MOVL C00416 V=800.0 PL=0
MOVL C00417 V=800.0 PL=0
MOVL C00418 V=800.0 PL=0
MOVL C00419 V=800.0 PL=0
MOVL C00420 V=800.0 PL=0
MOVL C00421 V=800.0 PL=0
MOVL C00422 V=800.0 PL=0
MOVL C00423 V=800.0 PL=0
MOVL C00424 V=800.0 PL=0
MOVL C00425 V=800.0 PL=0
MOVL C00426 V=800.0 PL=0
MOVL C00427 V=800.0 PL=0
MOVL C00428 V=800.0 PL=0
MOVL C00429 V=800.0 PL=0
MOVL C00430 V=800.0 PL=0
MOVL C00431 V=800.0 PL=0
MOVL C00432 V=800.0 PL=0
MOVL C00433 V=800.0 PL=0
MOVL C00434 V=800.0 PL=0
MOVL C00435 V=800.0 PL=0
MOVL C00436 V=800.0 PL=0
MOVL C00437 V=800.0 PL=0
MOVL C00438 V=800.0 PL=0
MOVL C00439 V=800.0 PL=0
MOVL C00440 V=800.0 PL=0
MOVL C00441 V=800.0 PL=0
MOVL C00442 V=800.0 PL=0
MOVL C00443 V=800.0 PL=0
MOVL C00444 V=800.0 PL=0
MOVL C00445 V=800.0 PL=0
MOVL C00446 V=800.0 PL=0
MOVL C00447 V=800.0 PL=0
MOVL C00448 V=800.0 PL=0
MOVL C00449 V=800.0 PL=0
MOVL C00450 V=800.0 PL=0
MOVL C00451 V=800.0 PL=0
MOVL C00452 V=800.0 PL=0
MOVL C00453 V=800.0 PL=0
MOVL C00454 V=800.0 PL=0
MOVL C00455 V=800.0 PL=0
MOVL C00456 V=800.0 PL=0
MOVL C00457 V=800.0 PL=0
MOVL C00458 V=800.0 PL=0
MOVL C00459 V=800.0 PL=0
MOVL C00460 V=800.0 PL=0
MOVL C00461 V=800.0 PL=0
MOVL C00462 V=800.0 PL=0
MOVL C00463 V=800.0 PL=0
MOVL C00464 V=800.0 PL=0
MOVL C00465 V=800.0 PL=0
MOVL C00466 V=800.0 PL=0
MOVL C00467 V=800.0 PL=0
MOVL C00468 V=800.0 PL=0
MOVL C00469 V=800.0 PL=0
MOVL C00470 V=800.0 PL=0
MOVL C00471 V=800.0 PL=0
MOVL C00472 V=800.0 PL=0
MOVL C00473 V=800.0 PL=0
MOVL C00474 V=800.0 PL=0
MOVL C00475 V=800.0 PL=0
MOVL C00476 V=800.0 PL=0
MOVL C00477 V=800.0 PL=0
MOVL C00478 V=800.0 PL=0
MOVL C00479 V=800.0 PL=0
MOVL C00480 V=800.0 PL=0
MOVL C00481 V=800.0 PL=0
MOVL C00482 V=800.0 PL=0
MOVL C00483 V=800.0 PL=0
MOVL C00484 V=800.0 PL=0
MOVL C00485 V=800.0 PL=0
MOVL C00486 V=800.0 PL=0
MOVL C00487 V=800.0 PL=0
MOVL C00488 V=800.0 PL=0
MOVL C00489 V=800.0 PL=0
MOVL C00490 V=800.0 PL=0
MOVL C00491 V=800.0 PL=0
MOVL C00492 V=800.0 PL=0
MOVL C00493 V=800.0 PL=0
MOVL C00494 V=800.0 PL=0
MOVL C00495 V=800.0 PL=0
MOVL C00496 V=800.0 PL=0
MOVL C00497 V=800.0 PL=0
MOVL C00498 V=800.0 PL=0
MOVL C00499 V=800.0 PL=0
MOVL C00500 V=800.0 PL=0
MOVL C00501 V=800.0 PL=0
MOVL C00502 V=800.0 PL=0
MOVL C00503 V=800.0 PL=0
MOVL C00504 V=800.0 PL=0
MOVL C00505 V=800.0 PL=0
MOVL C00506 V=800.0 PL=0
MOVL C00507 V=800.0 PL=0
MOVL C00508 V=800.0 PL=0
MOVL C00509 V=800.0 PL=0
MOVL C00510 V=800.0 PL=0
MOVL C00511 V=800.0 PL=0
MOVL C00512 V=800.0 PL=0
MOVL C00513 V=800.0 PL=0
MOVL C00514 V=800.0 PL=0
MOVL C00515 V=800.0 PL=0
MOVL C00516 V=800.0 PL=0
MOVL C00517 V=800.0 PL=0
MOVL C00518 V=800.0 PL=0
MOVL C00519 V=800.0 PL=0
MOVL C00520 V=800.0 PL=0
MOVL C00521 V=800.0 PL=0
MOVL C00522 V=800.0 PL=0
MOVL C00523 V=800.0 PL=0
MOVL C00524 V=800.0 PL=0
MOVL C00525 V=800.0 PL=0
MOVL C00526 V=800.0 PL=0
MOVL C00527 V=800.0 PL=0
MOVL C00528 V=800.0 PL=0
MOVL C00529 V=800.0 PL=0
MOVL C00530 V=800.0 PL=0
MOVL C00531 V=800.0 PL=0
MOVL C00532 V=800.0 PL=0
MOVL C00533 V=800.0 PL=0
MOVL C00534 V=800.0 PL=0
MOVL C00535 V=800.0 PL=0
MOVL C00536 V=800.0 PL=0
MOVL C00537 V=800.0 PL=0
MOVL C00538 V=800.0 PL=0
MOVL C00539 V=800.0 PL=0
MOVL C00540 V=800.0 PL=0
MOVL C00541 V=800.0 PL=0
MOVL C00542 V=800.0 PL=0
MOVL C00543 V=800.0 PL=0
MOVL C00544 V=800.0 PL=0
MOVL C00545 V=800.0 PL=0
MOVL C00546 V=800.0 PL=0
MOVL C00547 V=800.0 PL=0
MOVL C00548 V=800.0 PL=0
MOVL C00549 V=800.0 PL=0
MOVL C00550 V=800.0 PL=0
MOVL C00551 V=800.0 PL=0
MOVL C00552 V=800.0 PL=0
MOVL C00553 V=800.0 PL=0
MOVL C00554 V=800.0 PL=0
MOVL C00555 V=800.0 PL=0
MOVL C00556 V=800.0 PL=0
MOVL C00557 V=800.0 PL=0
MOVL C00558 V=800.0 PL=0
MOVL C00559 V=800.0 PL=0
MOVL C00560 V=800.0 PL=0
MOVL C00561 V=800.0 PL=0
MOVL C00562 V=800.0 PL=0
MOVL C00563 V=800.0 PL=0
MOVL C00564 V=800.0 PL=0
MOVL C00565 V=800.0 PL=0
MOVL C00566 V=800.0 PL=0
MOVL C00567 V=800.0 PL=0
MOVL C00568 V=800.0 PL=0
MOVL C00569 V=800.0 PL=0
MOVL C00570 V=800.0 PL=0
MOVL C00571 V=800.0 PL=0
MOVL C00572 V=800.0 PL=0
MOVL C00573 V=800.0 PL=0
MOVL C00574 V=800.0 PL=0
MOVL C00575 V=800.0 PL=0
MOVL C00576 V=800.0 PL=0
MOVL C00577 V=800.0 PL=0
MOVL C00578 V=800.0 PL=0
MOVL C00579 V=800.0 PL=0
MOVL C00580 V=800.0 PL=0
MOVL C00581 V=800.0 PL=0
MOVL C00582 V=800.0 PL=0
MOVL C00583 V=800.0 PL=0
MOVL C00584 V=800.0 PL=0
MOVL C00585 V=800.0 PL=0
MOVL C00586 V=800.0 PL=0
MOVL C00587 V=800.0 PL=0
MOVL C00588 V=800.0 PL=0
MOVL C00589 V=800.0 PL=0
MOVL C00590 V=800.0 PL=0
MOVL C00591 V=800.0 PL=0
MOVL C00592 V=800.0 PL=0
MOVL C00593 V=800.0 PL=0
MOVL C00594 V=800.0 PL=0
MOVL C00595 V=800.0 PL=0
MOVL C00596 V=800.0 PL=0
MOVL C00597 V=800.0 PL=0
MOVL C00598 V=800.0 PL=0
MOVL C00599 V=800.0 PL=0
MOVL C00600 V=800.0 PL=0
MOVL C00601 V=800.0 PL=0
MOVL C00602 V=800.0 PL=0
MOVL C00603 V=800.0 PL=0
MOVL C00604 V=800.0 PL=0
MOVL C00605 V=800.0 PL=0
MOVL C00606 V=800.0 PL=0
MOVL C00607 V=800.0 PL=0
MOVL C00608 V=800.0 PL=0
MOVL C00609 V=800.0 PL=0
MOVL C00610 V=800.0 PL=0
MOVL C00611 V=800.0 PL=0
MOVL C00612 V=800.0 PL=0
MOVL C00613 V=800.0 PL=0
MOVL C00614 V=800.0 PL=0
MOVL C00615 V=800.0 PL=0
MOVL C00616 V=800.0 PL=0
MOVL C00617 V=800.0 PL=0
MOVL C00618 V=800.0 PL=0
MOVL C00619 V=800.0 PL=0
MOVL C00620 V=800.0 PL=0
MOVL C00621 V=800.0 PL=0
MOVL C00622 V=800.0 PL=0
MOVL C00623 V=800.0 PL=0
MOVL C00624 V=800.0 PL=0
MOVL C00625 V=800.0 PL=0
MOVL C00626 V=800.0 PL=0
MOVL C00627 V=800.0 PL=0
MOVL C00628 V=800.0 PL=0
MOVL C00629 V=800.0 PL=0
MOVL C00630 V=800.0 PL=0
MOVL C00631 V=800.0 PL=0
MOVL C00632 V=800.0 PL=0
MOVL C00633 V=800.0 PL=0
MOVL C00634 V=800.0 PL=0
MOVL C00635 V=800.0 PL=0
MOVL C00636 V=800.0 PL=0
MOVL C00637 V=800.0 PL=0
MOVL C00638 V=800.0 PL=0
MOVL C00639 V=800.0 PL=0
MOVL C00640 V=800.0 PL=0
MOVL C00641 V=800.0 PL=0
MOVL C00642 V=800.0 PL=0
MOVL C00643 V=800.0 PL=0
MOVL C00644 V=800.0 PL=0
MOVL C00645 V=800.0 PL=0
MOVL C00646 V=800.0 PL=0
MOVL C00647 V=800.0 PL=0
MOVL C00648 V=800.0 PL=0
MOVL C00649 V=800.0 PL=0
MOVL C00650 V=800.0 PL=0
MOVL C00651 V=800.0 PL=0
MOVL C00652 V=800.0 PL=0
MOVL C00653 V=800.0 PL=0
MOVL C00654 V=800.0 PL=0
MOVL C00655 V=800.0 PL=0
MOVL C00656 V=800.0 PL=0
MOVL C00657 V=800.0 PL=0
MOVL C00658 V=800.0 PL=0
MOVL C00659 V=800.0 PL=0
MOVL C00660 V=800.0 PL=0
MOVL C00661 V=800.0 PL=0
MOVL C00662 V=800.0 PL=0
MOVL C00663 V=800.0 PL=0
MOVL C00664 V=800.0 PL=0
MOVL C00665 V=800.0 PL=0
MOVL C00666 V=800.0 PL=0
MOVL C00667 V=800.0 PL=0
MOVL C00668 V=800.0 PL=0
MOVL C00669 V=800.0 PL=0
MOVL C00670 V=800.0 PL=0
MOVL C00671 V=800.0 PL=0
MOVL C00672 V=800.0 PL=0
MOVL C00673 V=800.0 PL=0
MOVL C00674 V=800.0 PL=0
MOVL C00675 V=800.0 PL=0
MOVL C00676 V=800.0 PL=0
MOVL C00677 V=800.0 PL=0
MOVL C00678 V=800.0 PL=0
MOVL C00679 V=800.0 PL=0
MOVL C00680 V=800.0 PL=0
MOVL C00681 V=800.0 PL=0
MOVL C00682 V=800.0 PL=0
MOVL C00683 V=800.0 PL=0
MOVL C00684 V=800.0 PL=0
MOVL C00685 V=800.0 PL=0
MOVL C00686 V=800.0 PL=0
MOVL C00687 V=800.0 PL=0
MOVL C00688 V=800.0 PL=0
MOVL C00689 V=800.0 PL=0
MOVL C00690 V=800.0 PL=0
MOVL C00691 V=800.0 PL=0
MOVL C00692 V=800.0 PL=0
MOVL C00693 V=800.0 PL=0
MOVL C00694 V=800.0 PL=0
MOVL C00695 V=800.0 PL=0
MOVL C00696 V=800.0 PL=0
MOVL C00697 V=800.0 PL=0
MOVL C00698 V=800.0 PL=0
MOVL C00699 V=800.0 PL=0
MOVL C00700 V=800.0 PL=0
MOVL C00701 V=800.0 PL=0
MOVL C00702 V=800.0 PL=0
MOVL C00703 V=800.0 PL=0
MOVL C00704 V=800.0 PL=0
MOVL C00705 V=800.0 PL=0
MOVL C00706 V=800.0 PL=0
MOVL C00707 V=800.0 PL=0
MOVL C00708 V=800.0 PL=0
MOVL C00709 V=800.0 PL=0
MOVL C00710 V=800.0 PL=0
MOVL C00711 V=800.0 PL=0
MOVL C00712 V=800.0 PL=0
MOVL C00713 V=800.0 PL=0
MOVL C00714 V=800.0 PL=0
MOVL C00715 V=800.0 PL=0
MOVL C00716 V=800.0 PL=0
MOVL C00717 V=800.0 PL=0
MOVL C00718 V=800.0 PL=0
MOVL C00719 V=800.0 PL=0
MOVL C00720 V=800.0 PL=0
MOVL C00721 V=800.0 PL=0
MOVL C00722 V=800.0 PL=0
MOVL C00723 V=800.0 PL=0
MOVL C00724 V=800.0 PL=0
MOVL C00725 V=800.0 PL=0
MOVL C00726 V=800.0 PL=0
MOVL C00727 V=800.0 PL=0
MOVL C00728 V=800.0 PL=0
MOVL C00729 V=800.0 PL=0
MOVL C00730 V=800.0 PL=0
MOVL C00731 V=800.0 PL=0
MOVL C00732 V=800.0 PL=0
MOVL C00733 V=800.0 PL=0
MOVL C00734 V=800.0 PL=0
MOVL C00735 V=800.0 PL=0
MOVL C00736 V=800.0 PL=0
MOVL C00737 V=800.0 PL=0
MOVL C00738 V=800.0 PL=0
MOVL C00739 V=800.0 PL=0
MOVL C00740 V=800.0 PL=0
MOVL C00741 V=800.0 PL=0
MOVL C00742 V=800.0 PL=0
MOVL C00743 V=800.0 PL=0
MOVL C00744 V=800.0 PL=0
MOVL C00745 V=800.0 PL=0
MOVL C00746 V=800.0 PL=0
MOVL C00747 V=800.0 PL=0
MOVL C00748 V=800.0 PL=0
MOVL C00749 V=800.0 PL=0
MOVL C00750 V=800.0 PL=0
MOVL C00751 V=800.0 PL=0
MOVL C00752 V=800.0 PL=0
MOVL C00753 V=800.0 PL=0
MOVL C00754 V=800.0 PL=0
MOVL C00755 V=800.0 PL=0
MOVL C00756 V=800.0 PL=0
MOVL C00757 V=800.0 PL=0
MOVL C00758 V=800.0 PL=0
MOVL C00759 V=800.0 PL=0
MOVL C00760 V=800.0 PL=0
MOVL C00761 V=800.0 PL=0
MOVL C00762 V=800.0 PL=0
MOVL C00763 V=800.0 PL=0
MOVL C00764 V=800.0 PL=0
MOVL C00765 V=800.0 PL=0
MOVL C00766 V=800.0 PL=0
MOVL C00767 V=800.0 PL=0
MOVL C00768 V=800.0 PL=0
MOVL C00769 V=800.0 PL=0
MOVL C00770 V=800.0 PL=0
MOVL C00771 V=800.0 PL=0
MOVL C00772 V=800.0 PL=0
MOVL C00773 V=800.0 PL=0
MOVL C00774 V=800.0 PL=0
MOVL C00775 V=800.0 PL=0
MOVL C00776 V=800.0 PL=0
MOVL C00777 V=800.0 PL=0
MOVL C00778 V=800.0 PL=0
MOVL C00779 V=800.0 PL=0
MOVL C00780 V=800.0 PL=0
MOVL C00781 V=800.0 PL=0
MOVL C00782 V=800.0 PL=0
MOVL C00783 V=800.0 PL=0
MOVL C00784 V=800.0 PL=0
MOVL C00785 V=800.0 PL=0
MOVL C00786 V=800.0 PL=0
MOVL C00787 V=800.0 PL=0
MOVL C00788 V=800.0 PL=0
MOVL C00789 V=800.0 PL=0
MOVL C00790 V=800.0 PL=0
MOVL C00791 V=800.0 PL=0
MOVL C00792 V=800.0 PL=0
MOVL C00793 V=800.0 PL=0
MOVL C00794 V=800.0 PL=0
MOVL C00795 V=800.0 PL=0
MOVL C00796 V=800.0 PL=0
MOVL C00797 V=800.0 PL=0
MOVL C00798 V=800.0 PL=0
MOVL C00799 V=800.0 PL=0
MOVL C00800 V=800.0 PL=0
MOVL C00801 V=800.0 PL=0
MOVL C00802 V=800.0 PL=0
MOVL C00803 V=800.0 PL=0
MOVL C00804 V=800.0 PL=0
MOVL C00805 V=800.0 PL=0
MOVL C00806 V=800.0 PL=0
MOVL C00807 V=800.0 PL=0
MOVL C00808 V=800.0 PL=0
MOVL C00809 V=800.0 PL=0
MOVL C00810 V=800.0 PL=0
MOVL C00811 V=800.0 PL=0
MOVL C00812 V=800.0 PL=0
MOVL C00813 V=800.0 PL=0
MOVL C00814 V=800.0 PL=0
MOVL C00815 V=800.0 PL=0
MOVL C00816 V=800.0 PL=0
MOVL C00817 V=800.0 PL=0
MOVL C00818 V=800.0 PL=0
MOVL C00819 V=800.0 PL=0
MOVL C00820 V=800.0 PL=0
MOVL C00821 V=800.0 PL=0
MOVL C00822 V=800.0 PL=0
MOVL C00823 V=800.0 PL=0
MOVL C00824 V=800.0 PL=0
MOVL C00825 V=800.0 PL=0
MOVL C00826 V=800.0 PL=0
MOVL C00827 V=800.0 PL=0
MOVL C00828 V=800.0 PL=0
MOVL C00829 V=800.0 PL=0
MOVL C00830 V=800.0 PL=0
MOVL C00831 V=800.0 PL=0
MOVL C00832 V=800.0 PL=0
MOVL C00833 V=800.0 PL=0
MOVL C00834 V=800.0 PL=0
MOVL C00835 V=800.0 PL=0
MOVL C00836 V=800.0 PL=0
MOVL C00837 V=800.0 PL=0
MOVL C00838 V=800.0 PL=0
MOVL C00839 V=800.0 PL=0
MOVL C00840 V=800.0 PL=0
MOVL C00841 V=800.0 PL=0
MOVL C00842 V=800.0 PL=0
MOVL C00843 V=800.0 PL=0
MOVL C00844 V=800.0 PL=0
MOVL C00845 V=800.0 PL=0
MOVL C00846 V=800.0 PL=0
MOVL C00847 V=800.0 PL=0
MOVL C00848 V=800.0 PL=0
MOVL C00849 V=800.0 PL=0
MOVL C00850 V=800.0 PL=0
MOVL C00851 V=800.0 PL=0
MOVL C00852 V=800.0 PL=0
MOVL C00853 V=800.0 PL=0
MOVL C00854 V=800.0 PL=0
MOVL C00855 V=800.0 PL=0
MOVL C00856 V=800.0 PL=0
MOVL C00857 V=800.0 PL=0
MOVL C00858 V=800.0 PL=0
MOVL C00859 V=800.0 PL=0
MOVL C00860 V=800.0 PL=0
MOVL C00861 V=800.0 PL=0
MOVL C00862 V=800.0 PL=0
MOVL C00863 V=800.0 PL=0
MOVL C00864 V=800.0 PL=0
MOVL C00865 V=800.0 PL=0
MOVL C00866 V=800.0 PL=0
MOVL C00867 V=800.0 PL=0
MOVL C00868 V=800.0 PL=0
MOVL C00869 V=800.0 PL=0
MOVL C00870 V=800.0 PL=0
MOVL C00871 V=800.0 PL=0
MOVL C00872 V=800.0 PL=0
MOVL C00873 V=800.0 PL=0
MOVL C00874 V=800.0 PL=0
MOVL C00875 V=800.0 PL=0
MOVL C00876 V=800.0 PL=0
MOVL C00877 V=800.0 PL=0
MOVL C00878 V=800.0 PL=0
MOVL C00879 V=800.0 PL=0
MOVL C00880 V=800.0 PL=0
MOVL C00881 V=800.0 PL=0
MOVL C00882 V=800.0 PL=0
MOVL C00883 V=800.0 PL=0
MOVL C00884 V=800.0 PL=0
MOVL C00885 V=800.0 PL=0
MOVL C00886 V=800.0 PL=0
MOVL C00887 V=800.0 PL=0
MOVL C00888 V=800.0 PL=0
MOVL C00889 V=800.0 PL=0
MOVL C00890 V=800.0 PL=0
MOVL C00891 V=800.0 PL=0
MOVL C00892 V=800.0 PL=0
MOVL C00893 V=800.0 PL=0
MOVL C00894 V=800.0 PL=0
MOVL C00895 V=800.0 PL=0
MOVL C00896 V=800.0 PL=0
MOVL C00897 V=800.0 PL=0
MOVL C00898 V=800.0 PL=0
MOVL C00899 V=800.0 PL=0
MOVL C00900 V=800.0 PL=0
MOVL C00901 V=800.0 PL=0
MOVL C00902 V=800.0 PL=0
MOVL C00903 V=800.0 PL=0
MOVL C00904 V=800.0 PL=0
MOVL C00905 V=800.0 PL=0
MOVL C00906 V=800.0 PL=0
MOVL C00907 V=800.0 PL=0
MOVL C00908 V=800.0 PL=0
MOVL C00909 V=800.0 PL=0
MOVL C00910 V=800.0 PL=0
MOVL C00911 V=800.0 PL=0
MOVL C00912 V=800.0 PL=0
MOVL C00913 V=800.0 PL=0
MOVL C00914 V=800.0 PL=0
MOVL C00915 V=800.0 PL=0
MOVL C00916 V=800.0 PL=0
MOVL C00917 V=800.0 PL=0
MOVL C00918 V=800.0 PL=0
MOVL C00919 V=800.0 PL=0
MOVL C00920 V=800.0 PL=0
MOVL C00921 V=800.0 PL=0
MOVL C00922 V=800.0 PL=0
MOVL C00923 V=800.0 PL=0
MOVL C00924 V=800.0 PL=0
MOVL C00925 V=800.0 PL=0
MOVL C00926 V=800.0 PL=0
MOVL C00927 V=800.0 PL=0
MOVL C00928 V=800.0 PL=0
MOVL C00929 V=800.0 PL=0
MOVL C00930 V=800.0 PL=0
MOVL C00931 V=800.0 PL=0
MOVL C00932 V=800.0 PL=0
MOVL C00933 V=800.0 PL=0
MOVL C00934 V=800.0 PL=0
MOVL C00935 V=800.0 PL=0
MOVL C00936 V=800.0 PL=0
MOVL C00937 V=800.0 PL=0
MOVL C00938 V=800.0 PL=0
MOVL C00939 V=800.0 PL=0
MOVL C00940 V=800.0 PL=0
MOVL C00941 V=800.0 PL=0
MOVL C00942 V=800.0 PL=0
MOVL C00943 V=800.0 PL=0
MOVL C00944 V=800.0 PL=0
MOVL C00945 V=800.0 PL=0
MOVL C00946 V=800.0 PL=0
MOVL C00947 V=800.0 PL=0
MOVL C00948 V=800.0 PL=0
MOVL C00949 V=800.0 PL=0
MOVL C00950 V=800.0 PL=0
MOVL C00951 V=800.0 PL=0
MOVL C00952 V=800.0 PL=0
MOVL C00953 V=800.0 PL=0
MOVL C00954 V=800.0 PL=0
MOVL C00955 V=800.0 PL=0
MOVL C00956 V=800.0 PL=0
MOVL C00957 V=800.0 PL=0
MOVL C00958 V=800.0 PL=0
MOVL C00959 V=800.0 PL=0
MOVL C00960 V=800.0 PL=0
MOVL C00961 V=800.0 PL=0
MOVL C00962 V=800.0 PL=0
MOVL C00963 V=800.0 PL=0
MOVL C00964 V=800.0 PL=0
MOVL C00965 V=800.0 PL=0
MOVL C00966 V=800.0 PL=0
MOVL C00967 V=800.0 PL=0
MOVL C00968 V=800.0 PL=0
MOVL C00969 V=800.0 PL=0
MOVL C00970 V=800.0 PL=0
MOVL C00971 V=800.0 PL=0
MOVL C00972 V=800.0 PL=0
MOVL C00973 V=800.0 PL=0
MOVL C00974 V=800.0 PL=0
MOVL C00975 V=800.0 PL=0
MOVL C00976 V=800.0 PL=0
MOVL C00977 V=800.0 PL=0
MOVL C00978 V=800.0 PL=0
MOVL C00979 V=800.0 PL=0
MOVL C00980 V=800.0 PL=0
MOVL C00981 V=800.0 PL=0
MOVL C00982 V=800.0 PL=0
MOVL C00983 V=800.0 PL=0
MOVL C00984 V=800.0 PL=0
MOVL C00985 V=800.0 PL=0
MOVL C00986 V=800.0 PL=0
MOVL C00987 V=800.0 PL=0
MOVL C00988 V=800.0 PL=0
MOVL C00989 V=800.0 PL=0
MOVL C00990 V=800.0 PL=0
MOVL C00991 V=800.0 PL=0
MOVL C00992 V=800.0 PL=0
MOVL C00993 V=800.0 PL=0
MOVL C00994 V=800.0 PL=0
MOVL C00995 V=800.0 PL=0
MOVL C00996 V=800.0 PL=0
MOVL C00997 V=800.0 PL=0
MOVL C00998 V=800.0 PL=0
MOVL C00999 V=800.0 PL=0
MOVL C01000 V=800.0 PL=0
MOVL C01001 V=800.0 PL=0
MOVL C01002 V=800.0 PL=0
MOVL C01003 V=800.0 PL=0
MOVL C01004 V=800.0 PL=0
MOVL C01005 V=800.0 PL=0
MOVL C01006 V=800.0 PL=0
MOVL C01007 V=800.0 PL=0
MOVL C01008 V=800.0 PL=0
MOVL C01009 V=800.0 PL=0
MOVL C01010 V=800.0 PL=0
MOVL C01011 V=800.0 PL=0
MOVL C01012 V=800.0 PL=0
MOVL C01013 V=800.0 PL=0
MOVL C01014 V=800.0 PL=0
MOVL C01015 V=800.0 PL=0
MOVL C01016 V=800.0 PL=0
MOVL C01017 V=800.0 PL=0
MOVL C01018 V=800.0 PL=0
MOVL C01019 V=800.0 PL=0
MOVL C01020 V=800.0 PL=0
MOVL C01021 V=800.0 PL=0
MOVL C01022 V=800.0 PL=0
MOVL C01023 V=800.0 PL=0
MOVL C01024 V=800.0 PL=0
MOVL C01025 V=800.0 PL=0
MOVL C01026 V=800.0 PL=0
MOVL C01027 V=800.0 PL=0
MOVL C01028 V=800.0 PL=0
MOVL C01029 V=800.0 PL=0
MOVL C01030 V=800.0 PL=0
MOVL C01031 V=800.0 PL=0
MOVL C01032 V=800.0 PL=0
MOVL C01033 V=800.0 PL=0
MOVL C01034 V=800.0 PL=0
MOVL C01035 V=800.0 PL=0
MOVL C01036 V=800.0 PL=0
MOVL C01037 V=800.0 PL=0
MOVL C01038 V=800.0 PL=0
MOVL C01039 V=800.0 PL=0
MOVL C01040 V=800.0 PL=0
MOVL C01041 V=800.0 PL=0
MOVL C01042 V=800.0 PL=0
MOVL C01043 V=800.0 PL=0
MOVL C01044 V=800.0 PL=0
MOVL C01045 V=800.0 PL=0
MOVL C01046 V=800.0 PL=0
MOVL C01047 V=800.0 PL=0
MOVL C01048 V=800.0 PL=0
MOVL C01049 V=800.0 PL=0
MOVL C01050 V=800.0 PL=0
MOVL C01051 V=800.0 PL=0
MOVL C01052 V=800.0 PL=0
MOVL C01053 V=800.0 PL=0
MOVL C01054 V=800.0 PL=0
MOVL C01055 V=800.0 PL=0
MOVL C01056 V=800.0 PL=0
MOVL C01057 V=800.0 PL=0
MOVL C01058 V=800.0 PL=0
MOVL C01059 V=800.0 PL=0
MOVL C01060 V=800.0 PL=0
MOVL C01061 V=800.0 PL=0
MOVL C01062 V=800.0 PL=0
MOVL C01063 V=800.0 PL=0
MOVL C01064 V=800.0 PL=0
MOVL C01065 V=800.0 PL=0
MOVL C01066 V=800.0 PL=0
MOVL C01067 V=800.0 PL=0
MOVL C01068 V=800.0 PL=0
MOVL C01069 V=800.0 PL=0
MOVL C01070 V=800.0 PL=0
MOVL C01071 V=800.0 PL=0
MOVL C01072 V=800.0 PL=0
MOVL C01073 V=800.0 PL=0
MOVL C01074 V=800.0 PL=0
MOVL C01075 V=800.0 PL=0
MOVL C01076 V=800.0 PL=0
MOVL C01077 V=800.0 PL=0
MOVL C01078 V=800.0 PL=0
MOVL C01079 V=800.0 PL=0
MOVL C01080 V=800.0 PL=0
MOVL C01081 V=800.0 PL=0
MOVL C01082 V=800.0 PL=0
MOVL C01083 V=800.0 PL=0
MOVL C01084 V=800.0 PL=0
MOVL C01085 V=800.0 PL=0
MOVL C01086 V=800.0 PL=0
MOVL C01087 V=800.0 PL=0
MOVL C01088 V=800.0 PL=0
MOVL C01089 V=800.0 PL=0
MOVL C01090 V=800.0 PL=0
MOVL C01091 V=800.0 PL=0
MOVL C01092 V=800.0 PL=0
MOVL C01093 V=800.0 PL=0
MOVL C01094 V=800.0 PL=0
MOVL C01095 V=800.0 PL=0
MOVL C01096 V=800.0 PL=0
MOVL C01097 V=800.0 PL=0
MOVL C01098 V=800.0 PL=0
MOVL C01099 V=800.0 PL=0
MOVL C01100 V=800.0 PL=0
MOVL C01101 V=800.0 PL=0
MOVL C01102 V=800.0 PL=0
MOVL C01103 V=800.0 PL=0
MOVL C01104 V=800.0 PL=0
MOVL C01105 V=800.0 PL=0
MOVL C01106 V=800.0 PL=0
MOVL C01107 V=800.0 PL=0
MOVL C01108 V=800.0 PL=0
MOVL C01109 V=800.0 PL=0
MOVL C01110 V=800.0 PL=0
MOVL C01111 V=800.0 PL=0
MOVL C01112 V=800.0 PL=0
MOVL C01113 V=800.0 PL=0
MOVL C01114 V=800.0 PL=0
MOVL C01115 V=800.0 PL=0
MOVL C01116 V=800.0 PL=0
MOVL C01117 V=800.0 PL=0
MOVL C01118 V=800.0 PL=0
MOVL C01119 V=800.0 PL=0
MOVL C01120 V=800.0 PL=0
MOVL C01121 V=800.0 PL=0
MOVL C01122 V=800.0 PL=0
MOVL C01123 V=800.0 PL=0
MOVL C01124 V=800.0 PL=0
MOVL C01125 V=800.0 PL=0
MOVL C01126 V=800.0 PL=0
MOVL C01127 V=800.0 PL=0
MOVL C01128 V=800.0 PL=0
MOVL C01129 V=800.0 PL=0
MOVL C01130 V=800.0 PL=0
MOVL C01131 V=800.0 PL=0
MOVL C01132 V=800.0 PL=0
MOVL C01133 V=800.0 PL=0
MOVL C01134 V=800.0 PL=0
MOVL C01135 V=800.0 PL=0
MOVL C01136 V=800.0 PL=0
MOVL C01137 V=800.0 PL=0
MOVL C01138 V=800.0 PL=0
MOVL C01139 V=800.0 PL=0
MOVL C01140 V=800.0 PL=0
MOVL C01141 V=800.0 PL=0
MOVL C01142 V=800.0 PL=0
MOVL C01143 V=800.0 PL=0
MOVL C01144 V=800.0 PL=0
MOVL C01145 V=800.0 PL=0
MOVL C01146 V=800.0 PL=0
MOVL C01147 V=800.0 PL=0
MOVL C01148 V=800.0 PL=0
MOVL C01149 V=800.0 PL=0
MOVL C01150 V=800.0 PL=0
MOVL C01151 V=800.0 PL=0
MOVL C01152 V=800.0 PL=0
MOVL C01153 V=800.0 PL=0
MOVL C01154 V=800.0 PL=0
MOVL C01155 V=800.0 PL=0
MOVL C01156 V=800.0 PL=0
MOVL C01157 V=800.0 PL=0
MOVL C01158 V=800.0 PL=0
MOVL C01159 V=800.0 PL=0
MOVL C01160 V=800.0 PL=0
MOVL C01161 V=800.0 PL=0
MOVL C01162 V=800.0 PL=0
MOVL C01163 V=800.0 PL=0
MOVL C01164 V=800.0 PL=0
MOVL C01165 V=800.0 PL=0
MOVL C01166 V=800.0 PL=0
MOVL C01167 V=800.0 PL=0
MOVL C01168 V=800.0 PL=0
MOVL C01169 V=800.0 PL=0
MOVL C01170 V=800.0 PL=0
MOVL C01171 V=800.0 PL=0
MOVL C01172 V=800.0 PL=0
MOVL C01173 V=800.0 PL=0
MOVL C01174 V=800.0 PL=0
MOVL C01175 V=800.0 PL=0
MOVL C01176 V=800.0 PL=0
MOVL C01177 V=800.0 PL=0
MOVL C01178 V=800.0 PL=0
MOVL C01179 V=800.0 PL=0
MOVL C01180 V=800.0 PL=0
MOVL C01181 V=800.0 PL=0
MOVL C01182 V=800.0 PL=0
MOVL C01183 V=800.0 PL=0
MOVL C01184 V=800.0 PL=0
MOVL C01185 V=800.0 PL=0
MOVL C01186 V=800.0 PL=0
MOVL C01187 V=800.0 PL=0
MOVL C01188 V=800.0 PL=0
MOVL C01189 V=800.0 PL=0
MOVL C01190 V=800.0 PL=0
MOVL C01191 V=800.0 PL=0
MOVL C01192 V=800.0 PL=0
MOVL C01193 V=800.0 PL=0
MOVL C01194 V=800.0 PL=0
MOVL C01195 V=800.0 PL=0
MOVL C01196 V=800.0 PL=0
MOVL C01197 V=800.0 PL=0
MOVL C01198 V=800.0 PL=0
MOVL C01199 V=800.0 PL=0
MOVL C01200 V=800.0 PL=0
MOVL C01201 V=800.0 PL=0
MOVL C01202 V=800.0 PL=0
MOVL C01203 V=800.0 PL=0
MOVL C01204 V=800.0 PL=0
MOVL C01205 V=800.0 PL=0
MOVL C01206 V=800.0 PL=0
MOVL C01207 V=800.0 PL=0
MOVL C01208 V=800.0 PL=0
MOVL C01209 V=800.0 PL=0
MOVL C01210 V=800.0 PL=0
MOVL C01211 V=800.0 PL=0
MOVL C01212 V=800.0 PL=0
MOVL C01213 V=800.0 PL=0
MOVL C01214 V=800.0 PL=0
MOVL C01215 V=800.0 PL=0
MOVL C01216 V=800.0 PL=0
MOVL C01217 V=800.0 PL=0
MOVL C01218 V=800.0 PL=0
MOVL C01219 V=800.0 PL=0
MOVL C01220 V=800.0 PL=0
MOVL C01221 V=800.0 PL=0
MOVL C01222 V=800.0 PL=0
MOVL C01223 V=800.0 PL=0
MOVL C01224 V=800.0 PL=0
MOVL C01225 V=800.0 PL=0
MOVL C01226 V=800.0 PL=0
MOVL C01227 V=800.0 PL=0
MOVL C01228 V=800.0 PL=0
MOVL C01229 V=800.0 PL=0
MOVL C01230 V=800.0 PL=0
MOVL C01231 V=800.0 PL=0
MOVL C01232 V=800.0 PL=0
MOVL C01233 V=800.0 PL=0
MOVL C01234 V=800.0 PL=0
MOVL C01235 V=800.0 PL=0
MOVL C01236 V=800.0 PL=0
MOVL C01237 V=800.0 PL=0
MOVL C01238 V=800.0 PL=0
MOVL C01239 V=800.0 PL=0
MOVL C01240 V=800.0 PL=0
MOVL C01241 V=800.0 PL=0
MOVL C01242 V=800.0 PL=0
MOVL C01243 V=800.0 PL=0
MOVL C01244 V=800.0 PL=0
MOVL C01245 V=800.0 PL=0
MOVL C01246 V=800.0 PL=0
MOVL C01247 V=800.0 PL=0
MOVL C01248 V=800.0 PL=0
MOVL C01249 V=800.0 PL=0
MOVL C01250 V=800.0 PL=0
MOVL C01251 V=800.0 PL=0
MOVL C01252 V=800.0 PL=0
MOVL C01253 V=800.0 PL=0
MOVL C01254 V=800.0 PL=0
MOVL C01255 V=800.0 PL=0
MOVL C01256 V=800.0 PL=0
MOVL C01257 V=800.0 PL=0
MOVL C01258 V=800.0 PL=0
MOVL C01259 V=800.0 PL=0
MOVL C01260 V=800.0 PL=0
MOVL C01261 V=800.0 PL=0
MOVL C01262 V=800.0 PL=0
MOVL C01263 V=800.0 PL=0
MOVL C01264 V=800.0 PL=0
MOVL C01265 V=800.0 PL=0
MOVL C01266 V=800.0 PL=0
MOVL C01267 V=800.0 PL=0
MOVL C01268 V=800.0 PL=0
MOVL C01269 V=800.0 PL=0
MOVL C01270 V=800.0 PL=0
MOVL C01271 V=800.0 PL=0
MOVL C01272 V=800.0 PL=0
MOVL C01273 V=800.0 PL=0
MOVL C01274 V=800.0 PL=0
MOVL C01275 V=800.0 PL=0
MOVL C01276 V=800.0 PL=0
MOVL C01277 V=800.0 PL=0
MOVL C01278 V=800.0 PL=0
MOVL C01279 V=800.0 PL=0
MOVL C01280 V=800.0 PL=0
MOVL C01281 V=800.0 PL=0
MOVL C01282 V=800.0 PL=0
MOVL C01283 V=800.0 PL=0
MOVL C01284 V=800.0 PL=0
MOVL C01285 V=800.0 PL=0
MOVL C01286 V=800.0 PL=0
MOVL C01287 V=800.0 PL=0
MOVL C01288 V=800.0 PL=0
MOVL C01289 V=800.0 PL=0
MOVL C01290 V=800.0 PL=0
MOVL C01291 V=800.0 PL=0
MOVL C01292 V=800.0 PL=0
MOVL C01293 V=800.0 PL=0
MOVL C01294 V=800.0 PL=0
MOVL C01295 V=800.0 PL=0
MOVL C01296 V=800.0 PL=0
MOVL C01297 V=800.0 PL=0
MOVL C01298 V=800.0 PL=0
MOVL C01299 V=800.0 PL=0
MOVL C01300 V=800.0 PL=0
MOVL C01301 V=800.0 PL=0
MOVL C01302 V=800.0 PL=0
MOVL C01303 V=800.0 PL=0
MOVL C01304 V=800.0 PL=0
MOVL C01305 V=800.0 PL=0
MOVL C01306 V=800.0 PL=0
MOVL C01307 V=800.0 PL=0
MOVL C01308 V=800.0 PL=0
MOVL C01309 V=800.0 PL=0
MOVL C01310 V=800.0 PL=0
MOVL C01311 V=800.0 PL=0
MOVL C01312 V=800.0 PL=0
MOVL C01313 V=800.0 PL=0
MOVL C01314 V=800.0 PL=0
MOVL C01315 V=800.0 PL=0
MOVL C01316 V=800.0 PL=0
MOVL C01317 V=800.0 PL=0
MOVL C01318 V=800.0 PL=0
MOVL C01319 V=800.0 PL=0
MOVL C01320 V=800.0 PL=0
MOVL C01321 V=800.0 PL=0
MOVL C01322 V=800.0 PL=0
MOVL C01323 V=800.0 PL=0
MOVL C01324 V=800.0 PL=0
MOVL C01325 V=800.0 PL=0
MOVL C01326 V=800.0 PL=0
MOVL C01327 V=800.0 PL=0
MOVL C01328 V=800.0 PL=0
MOVL C01329 V=800.0 PL=0
MOVL C01330 V=800.0 PL=0
MOVL C01331 V=800.0 PL=0
MOVL C01332 V=800.0 PL=0
MOVL C01333 V=800.0 PL=0
MOVL C01334 V=800.0 PL=0
MOVL C01335 V=800.0 PL=0
MOVL C01336 V=800.0 PL=0
MOVL C01337 V=800.0 PL=0
MOVL C01338 V=800.0 PL=0
MOVL C01339 V=800.0 PL=0
MOVL C01340 V=800.0 PL=0
MOVL C01341 V=800.0 PL=0
MOVL C01342 V=800.0 PL=0
MOVL C01343 V=800.0 PL=0
MOVL C01344 V=800.0 PL=0
MOVL C01345 V=800.0 PL=0
MOVL C01346 V=800.0 PL=0
MOVL C01347 V=800.0 PL=0
MOVL C01348 V=800.0 PL=0
MOVL C01349 V=800.0 PL=0
MOVL C01350 V=800.0 PL=0
MOVL C01351 V=800.0 PL=0
MOVL C01352 V=800.0 PL=0
MOVL C01353 V=800.0 PL=0
MOVL C01354 V=800.0 PL=0
MOVL C01355 V=800.0 PL=0
MOVL C01356 V=800.0 PL=0
MOVL C01357 V=800.0 PL=0
MOVL C01358 V=800.0 PL=0
MOVL C01359 V=800.0 PL=0
MOVL C01360 V=800.0 PL=0
MOVL C01361 V=800.0 PL=0
MOVL C01362 V=800.0 PL=0
MOVL C01363 V=800.0 PL=0
MOVL C01364 V=800.0 PL=0
MOVL C01365 V=800.0 PL=0
MOVL C01366 V=800.0 PL=0
MOVL C01367 V=800.0 PL=0
MOVL C01368 V=800.0 PL=0
MOVL C01369 V=800.0 PL=0
MOVL C01370 V=800.0 PL=0
MOVL C01371 V=800.0 PL=0
MOVL C01372 V=800.0 PL=0
MOVL C01373 V=800.0 PL=0
MOVL C01374 V=800.0 PL=0
MOVL C01375 V=800.0 PL=0
MOVL C01376 V=800.0 PL=0
MOVL C01377 V=800.0 PL=0
MOVL C01378 V=800.0 PL=0
MOVL C01379 V=800.0 PL=0
MOVL C01380 V=800.0 PL=0
MOVL C01381 V=800.0 PL=0
MOVL C01382 V=800.0 PL=0
MOVL C01383 V=800.0 PL=0
MOVL C01384 V=800.0 PL=0
MOVL C01385 V=800.0 PL=0
MOVL C01386 V=800.0 PL=0
MOVL C01387 V=800.0 PL=0
MOVL C01388 V=800.0 PL=0
MOVL C01389 V=800.0 PL=0
MOVL C01390 V=800.0 PL=0
MOVL C01391 V=800.0 PL=0
MOVL C01392 V=800.0 PL=0
MOVL C01393 V=800.0 PL=0
MOVL C01394 V=800.0 PL=0
MOVL C01395 V=800.0 PL=0
MOVL C01396 V=800.0 PL=0
MOVL C01397 V=800.0 PL=0
MOVL C01398 V=800.0 PL=0
MOVL C01399 V=800.0 PL=0
MOVL C01400 V=800.0 PL=0
MOVL C01401 V=800.0 PL=0
MOVL C01402 V=800.0 PL=0
MOVL C01403 V=800.0 PL=0
MOVL C01404 V=800.0 PL=0
MOVL C01405 V=800.0 PL=0
MOVL C01406 V=800.0 PL=0
MOVL C01407 V=800.0 PL=0
MOVL C01408 V=800.0 PL=0
MOVL C01409 V=800.0 PL=0
MOVL C01410 V=800.0 PL=0
MOVL C01411 V=800.0 PL=0
MOVL C01412 V=800.0 PL=0
MOVL C01413 V=800.0 PL=0
MOVL C01414 V=800.0 PL=0
MOVL C01415 V=800.0 PL=0
MOVL C01416 V=800.0 PL=0
MOVL C01417 V=800.0 PL=0
MOVL C01418 V=800.0 PL=0
MOVL C01419 V=800.0 PL=0
MOVL C01420 V=800.0 PL=0
MOVL C01421 V=800.0 PL=0
MOVL C01422 V=800.0 PL=0
MOVL C01423 V=800.0 PL=0
MOVL C01424 V=800.0 PL=0
MOVL C01425 V=800.0 PL=0
MOVL C01426 V=800.0 PL=0
MOVL C01427 V=800.0 PL=0
MOVL C01428 V=800.0 PL=0
MOVL C01429 V=800.0 PL=0
MOVL C01430 V=800.0 PL=0
MOVL C01431 V=800.0 PL=0
MOVL C01432 V=800.0 PL=0
MOVL C01433 V=800.0 PL=0
MOVL C01434 V=800.0 PL=0
MOVL C01435 V=800.0 PL=0
MOVL C01436 V=800.0 PL=0
MOVL C01437 V=800.0 PL=0
MOVL C01438 V=800.0 PL=0
MOVL C01439 V=800.0 PL=0
MOVL C01440 V=800.0 PL=0
MOVL C01441 V=800.0 PL=0
MOVL C01442 V=800.0 PL=0
MOVL C01443 V=800.0 PL=0
MOVL C01444 V=800.0 PL=0
MOVL C01445 V=800.0 PL=0
MOVL C01446 V=800.0 PL=0
MOVL C01447 V=800.0 PL=0
MOVL C01448 V=800.0 PL=0
MOVL C01449 V=800.0 PL=0
MOVL C01450 V=800.0 PL=0
MOVL C01451 V=800.0 PL=0
MOVL C01452 V=800.0 PL=0
MOVL C01453 V=800.0 PL=0
MOVL C01454 V=800.0 PL=0
MOVL C01455 V=800.0 PL=0
MOVL C01456 V=800.0 PL=0
MOVL C01457 V=800.0 PL=0
MOVL C01458 V=800.0 PL=0
MOVL C01459 V=800.0 PL=0
MOVL C01460 V=800.0 PL=0
MOVL C01461 V=800.0 PL=0
MOVL C01462 V=800.0 PL=0
MOVL C01463 V=800.0 PL=0
MOVL C01464 V=800.0 PL=0
MOVL C01465 V=800.0 PL=0
MOVL C01466 V=800.0 PL=0
MOVL C01467 V=800.0 PL=0
MOVL C01468 V=800.0 PL=0
MOVL C01469 V=800.0 PL=0
MOVL C01470 V=800.0 PL=0
MOVL C01471 V=800.0 PL=0
MOVL C01472 V=800.0 PL=0
MOVL C01473 V=800.0 PL=0
MOVL C01474 V=800.0 PL=0
MOVL C01475 V=800.0 PL=0
MOVL C01476 V=800.0 PL=0
MOVL C01477 V=800.0 PL=0
MOVL C01478 V=800.0 PL=0
MOVL C01479 V=800.0 PL=0
MOVL C01480 V=800.0 PL=0
MOVL C01481 V=800.0 PL=0
MOVL C01482 V=800.0 PL=0
MOVL C01483 V=800.0 PL=0
MOVL C01484 V=800.0 PL=0
MOVL C01485 V=800.0 PL=0
MOVL C01486 V=800.0 PL=0
MOVL C01487 V=800.0 PL=0
MOVL C01488 V=800.0 PL=0
MOVL C01489 V=800.0 PL=0
MOVL C01490 V=800.0 PL=0
MOVL C01491 V=800.0 PL=0
MOVL C01492 V=800.0 PL=0
MOVL C01493 V=800.0 PL=0
MOVL C01494 V=800.0 PL=0
MOVL C01495 V=800.0 PL=0
MOVL C01496 V=800.0 PL=0
MOVL C01497 V=800.0 PL=0
MOVL C01498 V=800.0 PL=0
MOVL C01499 V=800.0 PL=0
MOVL C01500 V=800.0 PL=0
MOVL C01501 V=800.0 PL=0
MOVL C01502 V=800.0 PL=0
MOVL C01503 V=800.0 PL=0
MOVL C01504 V=800.0 PL=0
MOVL C01505 V=800.0 PL=0
MOVL C01506 V=800.0 PL=0
MOVL C01507 V=800.0 PL=0
MOVL C01508 V=800.0 PL=0
MOVL C01509 V=800.0 PL=0
MOVL C01510 V=800.0 PL=0
MOVL C01511 V=800.0 PL=0
MOVL C01512 V=800.0 PL=0
MOVL C01513 V=800.0 PL=0
MOVL C01514 V=800.0 PL=0
MOVL C01515 V=800.0 PL=0
MOVL C01516 V=800.0 PL=0
MOVL C01517 V=800.0 PL=0
MOVL C01518 V=800.0 PL=0
MOVL C01519 V=800.0 PL=0
MOVL C01520 V=800.0 PL=0
MOVL C01521 V=800.0 PL=0
MOVL C01522 V=800.0 PL=0
MOVL C01523 V=800.0 PL=0
MOVL C01524 V=800.0 PL=0
MOVL C01525 V=800.0 PL=0
MOVL C01526 V=800.0 PL=0
MOVL C01527 V=800.0 PL=0
MOVL C01528 V=800.0 PL=0
MOVL C01529 V=800.0 PL=0
MOVL C01530 V=800.0 PL=0
MOVL C01531 V=800.0 PL=0
MOVL C01532 V=800.0 PL=0
MOVL C01533 V=800.0 PL=0
MOVL C01534 V=800.0 PL=0
MOVL C01535 V=800.0 PL=0
MOVL C01536 V=800.0 PL=0
MOVL C01537 V=800.0 PL=0
MOVL C01538 V=800.0 PL=0
MOVL C01539 V=800.0 PL=0
MOVL C01540 V=800.0 PL=0
MOVL C01541 V=800.0 PL=0
MOVL C01542 V=800.0 PL=0
MOVL C01543 V=800.0 PL=0
MOVL C01544 V=800.0 PL=0
MOVL C01545 V=800.0 PL=0
MOVL C01546 V=800.0 PL=0
MOVL C01547 V=800.0 PL=0
MOVL C01548 V=800.0 PL=0
MOVL C01549 V=800.0 PL=0
MOVL C01550 V=800.0 PL=0
MOVL C01551 V=800.0 PL=0
MOVL C01552 V=800.0 PL=0
MOVL C01553 V=800.0 PL=0
MOVL C01554 V=800.0 PL=0
MOVL C01555 V=800.0 PL=0
MOVL C01556 V=800.0 PL=0
MOVL C01557 V=800.0 PL=0
MOVL C01558 V=800.0 PL=0
MOVL C01559 V=800.0 PL=0
MOVL C01560 V=800.0 PL=0
MOVL C01561 V=800.0 PL=0
MOVL C01562 V=800.0 PL=0
MOVL C01563 V=800.0 PL=0
MOVL C01564 V=800.0 PL=0
MOVL C01565 V=800.0 PL=0
MOVL C01566 V=800.0 PL=0
MOVL C01567 V=800.0 PL=0
MOVL C01568 V=800.0 PL=0
MOVL C01569 V=800.0 PL=0
MOVL C01570 V=800.0 PL=0
MOVL C01571 V=800.0 PL=0
MOVL C01572 V=800.0 PL=0
MOVL C01573 V=800.0 PL=0
MOVL C01574 V=800.0 PL=0
MOVL C01575 V=800.0 PL=0
MOVL C01576 V=800.0 PL=0
MOVL C01577 V=800.0 PL=0
MOVL C01578 V=800.0 PL=0
MOVL C01579 V=800.0 PL=0
MOVL C01580 V=800.0 PL=0
MOVL C01581 V=800.0 PL=0
MOVL C01582 V=800.0 PL=0
MOVL C01583 V=800.0 PL=0
MOVL C01584 V=800.0 PL=0
MOVL C01585 V=800.0 PL=0
MOVL C01586 V=800.0 PL=0
MOVL C01587 V=800.0 PL=0
MOVL C01588 V=800.0 PL=0
MOVL C01589 V=800.0 PL=0
MOVL C01590 V=800.0 PL=0
MOVL C01591 V=800.0 PL=0
MOVL C01592 V=800.0 PL=0
MOVL C01593 V=800.0 PL=0
MOVL C01594 V=800.0 PL=0
MOVL C01595 V=800.0 PL=0
MOVL C01596 V=800.0 PL=0
MOVL C01597 V=800.0 PL=0
MOVL C01598 V=800.0 PL=0
MOVL C01599 V=800.0 PL=0
MOVL C01600 V=800.0 PL=0
MOVL C01601 V=800.0 PL=0
MOVL C01602 V=800.0 PL=0
MOVL C01603 V=800.0 PL=0
MOVL C01604 V=800.0 PL=0
MOVL C01605 V=800.0 PL=0
MOVL C01606 V=800.0 PL=0
MOVL C01607 V=800.0 PL=0
MOVL C01608 V=800.0 PL=0
MOVL C01609 V=800.0 PL=0
MOVL C01610 V=800.0 PL=0
MOVL C01611 V=800.0 PL=0
MOVL C01612 V=800.0 PL=0
MOVL C01613 V=800.0 PL=0
MOVL C01614 V=800.0 PL=0
MOVL C01615 V=800.0 PL=0
MOVL C01616 V=800.0 PL=0
MOVL C01617 V=800.0 PL=0
MOVL C01618 V=800.0 PL=0
MOVL C01619 V=800.0 PL=0
MOVL C01620 V=800.0 PL=0
MOVL C01621 V=800.0 PL=0
MOVL C01622 V=800.0 PL=0
MOVL C01623 V=800.0 PL=0
MOVL C01624 V=800.0 PL=0
MOVL C01625 V=800.0 PL=0
MOVL C01626 V=800.0 PL=0
MOVL C01627 V=800.0 PL=0
MOVL C01628 V=800.0 PL=0
MOVL C01629 V=800.0 PL=0
MOVL C01630 V=800.0 PL=0
MOVL C01631 V=800.0 PL=0
MOVL C01632 V=800.0 PL=0
MOVL C01633 V=800.0 PL=0
MOVL C01634 V=800.0 PL=0
MOVL C01635 V=800.0 PL=0
MOVL C01636 V=800.0 PL=0
MOVL C01637 V=800.0 PL=0
MOVL C01638 V=800.0 PL=0
MOVL C01639 V=800.0 PL=0
MOVL C01640 V=800.0 PL=0
MOVL C01641 V=800.0 PL=0
MOVL C01642 V=800.0 PL=0
MOVL C01643 V=800.0 PL=0
MOVL C01644 V=800.0 PL=0
MOVL C01645 V=800.0 PL=0
MOVL C01646 V=800.0 PL=0
MOVL C01647 V=800.0 PL=0
MOVL C01648 V=800.0 PL=0
MOVL C01649 V=800.0 PL=0
MOVL C01650 V=800.0 PL=0
MOVL C01651 V=800.0 PL=0
MOVL C01652 V=800.0 PL=0
MOVL C01653 V=800.0 PL=0
MOVL C01654 V=800.0 PL=0
MOVL C01655 V=800.0 PL=0
MOVL C01656 V=800.0 PL=0
MOVL C01657 V=800.0 PL=0
MOVL C01658 V=800.0 PL=0
MOVL C01659 V=800.0 PL=0
MOVL C01660 V=800.0 PL=0
MOVL C01661 V=800.0 PL=0
MOVL C01662 V=800.0 PL=0
MOVL C01663 V=800.0 PL=0
MOVL C01664 V=800.0 PL=0
MOVL C01665 V=800.0 PL=0
MOVL C01666 V=800.0 PL=0
MOVL C01667 V=800.0 PL=0
MOVL C01668 V=800.0 PL=0
MOVL C01669 V=800.0 PL=0
MOVL C01670 V=800.0 PL=0
MOVL C01671 V=800.0 PL=0
MOVL C01672 V=800.0 PL=0
MOVL C01673 V=800.0 PL=0
MOVL C01674 V=800.0 PL=0
MOVL C01675 V=800.0 PL=0
MOVL C01676 V=800.0 PL=0
MOVL C01677 V=800.0 PL=0
MOVL C01678 V=800.0 PL=0
MOVL C01679 V=800.0 PL=0
MOVL C01680 V=800.0 PL=0
MOVL C01681 V=800.0 PL=0
MOVL C01682 V=800.0 PL=0
MOVL C01683 V=800.0 PL=0
MOVL C01684 V=800.0 PL=0
MOVL C01685 V=800.0 PL=0
MOVL C01686 V=800.0 PL=0
MOVL C01687 V=800.0 PL=0
MOVL C01688 V=800.0 PL=0
MOVL C01689 V=800.0 PL=0
MOVL C01690 V=800.0 PL=0
MOVL C01691 V=800.0 PL=0
MOVL C01692 V=800.0 PL=0
MOVL C01693 V=800.0 PL=0
MOVL C01694 V=800.0 PL=0
MOVL C01695 V=800.0 PL=0
MOVL C01696 V=800.0 PL=0
MOVL C01697 V=800.0 PL=0
MOVL C01698 V=800.0 PL=0
MOVL C01699 V=800.0 PL=0
MOVL C01700 V=800.0 PL=0
MOVL C01701 V=800.0 PL=0
MOVL C01702 V=800.0 PL=0
MOVL C01703 V=800.0 PL=0
MOVL C01704 V=800.0 PL=0
MOVL C01705 V=800.0 PL=0
MOVL C01706 V=800.0 PL=0
MOVL C01707 V=800.0 PL=0
MOVL C01708 V=800.0 PL=0
MOVL C01709 V=800.0 PL=0
MOVL C01710 V=800.0 PL=0
MOVL C01711 V=800.0 PL=0
MOVL C01712 V=800.0 PL=0
MOVL C01713 V=800.0 PL=0
MOVL C01714 V=800.0 PL=0
MOVL C01715 V=800.0 PL=0
MOVL C01716 V=800.0 PL=0
MOVL C01717 V=800.0 PL=0
MOVL C01718 V=800.0 PL=0
MOVL C01719 V=800.0 PL=0
MOVL C01720 V=800.0 PL=0
MOVL C01721 V=800.0 PL=0
MOVL C01722 V=800.0 PL=0
MOVL C01723 V=800.0 PL=0
MOVL C01724 V=800.0 PL=0
MOVL C01725 V=800.0 PL=0
MOVL C01726 V=800.0 PL=0
MOVL C01727 V=800.0 PL=0
MOVL C01728 V=800.0 PL=0
MOVL C01729 V=800.0 PL=0
MOVL C01730 V=800.0 PL=0
MOVL C01731 V=800.0 PL=0
MOVL C01732 V=800.0 PL=0
MOVL C01733 V=800.0 PL=0
MOVL C01734 V=800.0 PL=0
MOVL C01735 V=800.0 PL=0
MOVL C01736 V=800.0 PL=0
MOVL C01737 V=800.0 PL=0
MOVL C01738 V=800.0 PL=0
MOVL C01739 V=800.0 PL=0
MOVL C01740 V=800.0 PL=0
MOVL C01741 V=800.0 PL=0
MOVL C01742 V=800.0 PL=0
MOVL C01743 V=800.0 PL=0
MOVL C01744 V=800.0 PL=0
MOVL C01745 V=800.0 PL=0
MOVL C01746 V=800.0 PL=0
MOVL C01747 V=800.0 PL=0
MOVL C01748 V=800.0 PL=0
MOVL C01749 V=800.0 PL=0
MOVL C01750 V=800.0 PL=0
MOVL C01751 V=800.0 PL=0
MOVL C01752 V=800.0 PL=0
MOVL C01753 V=800.0 PL=0
MOVL C01754 V=800.0 PL=0
MOVL C01755 V=800.0 PL=0
MOVL C01756 V=800.0 PL=0
MOVL C01757 V=800.0 PL=0
MOVL C01758 V=800.0 PL=0
MOVL C01759 V=800.0 PL=0
MOVL C01760 V=800.0 PL=0
MOVL C01761 V=800.0 PL=0
MOVL C01762 V=800.0 PL=0
MOVL C01763 V=800.0 PL=0
MOVL C01764 V=800.0 PL=0
MOVL C01765 V=800.0 PL=0
MOVL C01766 V=800.0 PL=0
MOVL C01767 V=800.0 PL=0
MOVL C01768 V=800.0 PL=0
MOVL C01769 V=800.0 PL=0
MOVL C01770 V=800.0 PL=0
MOVL C01771 V=800.0 PL=0
MOVL C01772 V=800.0 PL=0
MOVL C01773 V=800.0 PL=0
MOVL C01774 V=800.0 PL=0
MOVL C01775 V=800.0 PL=0
MOVL C01776 V=800.0 PL=0
MOVL C01777 V=800.0 PL=0
MOVL C01778 V=800.0 PL=0
MOVL C01779 V=800.0 PL=0
MOVL C01780 V=800.0 PL=0
MOVL C01781 V=800.0 PL=0
MOVL C01782 V=800.0 PL=0
MOVL C01783 V=800.0 PL=0
MOVL C01784 V=800.0 PL=0
MOVL C01785 V=800.0 PL=0
MOVL C01786 V=800.0 PL=0
MOVL C01787 V=800.0 PL=0
MOVL C01788 V=800.0 PL=0
MOVL C01789 V=800.0 PL=0
MOVL C01790 V=800.0 PL=0
MOVL C01791 V=800.0 PL=0
MOVL C01792 V=800.0 PL=0
MOVL C01793 V=800.0 PL=0
MOVL C01794 V=800.0 PL=0
MOVL C01795 V=800.0 PL=0
MOVL C01796 V=800.0 PL=0
MOVL C01797 V=800.0 PL=0
MOVL C01798 V=800.0 PL=0
MOVL C01799 V=800.0 PL=0
MOVL C01800 V=800.0 PL=0
MOVL C01801 V=800.0 PL=0
MOVL C01802 V=800.0 PL=0
MOVL C01803 V=800.0 PL=0
MOVL C01804 V=800.0 PL=0
MOVL C01805 V=800.0 PL=0
MOVL C01806 V=800.0 PL=0
MOVL C01807 V=800.0 PL=0
MOVL C01808 V=800.0 PL=0
MOVL C01809 V=800.0 PL=0
MOVL C01810 V=800.0 PL=0
MOVL C01811 V=800.0 PL=0
MOVL C01812 V=800.0 PL=0
MOVL C01813 V=800.0 PL=0
MOVL C01814 V=800.0 PL=0
MOVL C01815 V=800.0 PL=0
MOVL C01816 V=800.0 PL=0
MOVL C01817 V=800.0 PL=0
MOVL C01818 V=800.0 PL=0
MOVL C01819 V=800.0 PL=0
MOVL C01820 V=800.0 PL=0
MOVL C01821 V=800.0 PL=0
MOVL C01822 V=800.0 PL=0
MOVL C01823 V=800.0 PL=0
MOVL C01824 V=800.0 PL=0
MOVL C01825 V=800.0 PL=0
MOVL C01826 V=800.0 PL=0
MOVL C01827 V=800.0 PL=0
MOVL C01828 V=800.0 PL=0
MOVL C01829 V=800.0 PL=0
MOVL C01830 V=800.0 PL=0
MOVL C01831 V=800.0 PL=0
MOVL C01832 V=800.0 PL=0
MOVL C01833 V=800.0 PL=0
MOVL C01834 V=800.0 PL=0
MOVL C01835 V=800.0 PL=0
MOVL C01836 V=800.0 PL=0
MOVL C01837 V=800.0 PL=0
MOVL C01838 V=800.0 PL=0
MOVL C01839 V=800.0 PL=0
MOVL C01840 V=800.0 PL=0
MOVL C01841 V=800.0 PL=0
MOVL C01842 V=800.0 PL=0
MOVL C01843 V=800.0 PL=0
MOVL C01844 V=800.0 PL=0
MOVL C01845 V=800.0 PL=0
MOVL C01846 V=800.0 PL=0
MOVL C01847 V=800.0 PL=0
MOVL C01848 V=800.0 PL=0
MOVL C01849 V=800.0 PL=0
MOVL C01850 V=800.0 PL=0
MOVL C01851 V=800.0 PL=0
MOVL C01852 V=800.0 PL=0
MOVL C01853 V=800.0 PL=0
MOVL C01854 V=800.0 PL=0
MOVL C01855 V=800.0 PL=0
MOVL C01856 V=800.0 PL=0
MOVL C01857 V=800.0 PL=0
MOVL C01858 V=800.0 PL=0
MOVL C01859 V=800.0 PL=0
MOVL C01860 V=800.0 PL=0
MOVL C01861 V=800.0 PL=0
MOVL C01862 V=800.0 PL=0
MOVL C01863 V=800.0 PL=0
MOVL C01864 V=800.0 PL=0
MOVL C01865 V=800.0 PL=0
MOVL C01866 V=800.0 PL=0
MOVL C01867 V=800.0 PL=0
MOVL C01868 V=800.0 PL=0
MOVL C01869 V=800.0 PL=0
MOVL C01870 V=800.0 PL=0
MOVL C01871 V=800.0 PL=0
MOVL C01872 V=800.0 PL=0
MOVL C01873 V=800.0 PL=0
MOVL C01874 V=800.0 PL=0
MOVL C01875 V=800.0 PL=0
MOVL C01876 V=800.0 PL=0
MOVL C01877 V=800.0 PL=0
MOVL C01878 V=800.0 PL=0
MOVL C01879 V=800.0 PL=0
MOVL C01880 V=800.0 PL=0
MOVL C01881 V=800.0 PL=0
MOVL C01882 V=800.0 PL=0
MOVL C01883 V=800.0 PL=0
MOVL C01884 V=800.0 PL=0
MOVL C01885 V=800.0 PL=0
MOVL C01886 V=800.0 PL=0
MOVL C01887 V=800.0 PL=0
MOVL C01888 V=800.0 PL=0
MOVL C01889 V=800.0 PL=0
MOVL C01890 V=800.0 PL=0
MOVL C01891 V=800.0 PL=0
MOVL C01892 V=800.0 PL=0
MOVL C01893 V=800.0 PL=0
MOVL C01894 V=800.0 PL=0
MOVL C01895 V=800.0 PL=0
MOVL C01896 V=800.0 PL=0
MOVL C01897 V=800.0 PL=0
MOVL C01898 V=800.0 PL=0
MOVL C01899 V=800.0 PL=0
MOVL C01900 V=800.0 PL=0
MOVL C01901 V=800.0 PL=0
MOVL C01902 V=800.0 PL=0
MOVL C01903 V=800.0 PL=0
MOVL C01904 V=800.0 PL=0
MOVL C01905 V=800.0 PL=0
MOVL C01906 V=800.0 PL=0
MOVL C01907 V=800.0 PL=0
MOVL C01908 V=800.0 PL=0
MOVL C01909 V=800.0 PL=0
MOVL C01910 V=800.0 PL=0
MOVL C01911 V=800.0 PL=0
MOVL C01912 V=800.0 PL=0
MOVL C01913 V=800.0 PL=0
MOVL C01914 V=800.0 PL=0
MOVL C01915 V=800.0 PL=0
MOVL C01916 V=800.0 PL=0
MOVL C01917 V=800.0 PL=0
MOVL C01918 V=800.0 PL=0
MOVL C01919 V=800.0 PL=0
MOVL C01920 V=800.0 PL=0
MOVL C01921 V=800.0 PL=0
MOVL C01922 V=800.0 PL=0
MOVL C01923 V=800.0 PL=0
MOVL C01924 V=800.0 PL=0
MOVL C01925 V=800.0 PL=0
MOVL C01926 V=800.0 PL=0
MOVL C01927 V=800.0 PL=0
MOVL C01928 V=800.0 PL=0
MOVL C01929 V=800.0 PL=0
MOVL C01930 V=800.0 PL=0
MOVL C01931 V=800.0 PL=0
MOVL C01932 V=800.0 PL=0
MOVL C01933 V=800.0 PL=0
MOVL C01934 V=800.0 PL=0
MOVL C01935 V=800.0 PL=0
MOVL C01936 V=800.0 PL=0
MOVL C01937 V=800.0 PL=0
MOVL C01938 V=800.0 PL=0
MOVL C01939 V=800.0 PL=0
MOVL C01940 V=800.0 PL=0
MOVL C01941 V=800.0 PL=0
MOVL C01942 V=800.0 PL=0
MOVL C01943 V=800.0 PL=0
MOVL C01944 V=800.0 PL=0
MOVL C01945 V=800.0 PL=0
MOVL C01946 V=800.0 PL=0
MOVL C01947 V=800.0 PL=0
MOVL C01948 V=800.0 PL=0
MOVL C01949 V=800.0 PL=0
MOVL C01950 V=800.0 PL=0
MOVL C01951 V=800.0 PL=0
MOVL C01952 V=800.0 PL=0
MOVL C01953 V=800.0 PL=0
MOVL C01954 V=800.0 PL=0
MOVL C01955 V=800.0 PL=0
MOVL C01956 V=800.0 PL=0
MOVL C01957 V=800.0 PL=0
MOVL C01958 V=800.0 PL=0
MOVL C01959 V=800.0 PL=0
MOVL C01960 V=800.0 PL=0
MOVL C01961 V=800.0 PL=0
MOVL C01962 V=800.0 PL=0
MOVL C01963 V=800.0 PL=0
MOVL C01964 V=800.0 PL=0
MOVL C01965 V=800.0 PL=0
MOVL C01966 V=800.0 PL=0
MOVL C01967 V=800.0 PL=0
MOVL C01968 V=800.0 PL=0
MOVL C01969 V=800.0 PL=0
MOVL C01970 V=800.0 PL=0
MOVL C01971 V=800.0 PL=0
MOVL C01972 V=800.0 PL=0
MOVL C01973 V=800.0 PL=0
MOVL C01974 V=800.0 PL=0
MOVL C01975 V=800.0 PL=0
MOVL C01976 V=800.0 PL=0
MOVL C01977 V=800.0 PL=0
MOVL C01978 V=800.0 PL=0
MOVL C01979 V=800.0 PL=0
MOVL C01980 V=800.0 PL=0
MOVL C01981 V=800.0 PL=0
MOVL C01982 V=800.0 PL=0
MOVL C01983 V=800.0 PL=0
MOVL C01984 V=800.0 PL=0
MOVL C01985 V=800.0 PL=0
MOVL C01986 V=800.0 PL=0
MOVL C01987 V=800.0 PL=0
MOVL C01988 V=800.0 PL=0
MOVL C01989 V=800.0 PL=0
MOVL C01990 V=800.0 PL=0
MOVL C01991 V=800.0 PL=0
MOVL C01992 V=800.0 PL=0
MOVL C01993 V=800.0 PL=0
MOVL C01994 V=800.0 PL=0
MOVL C01995 V=800.0 PL=0
MOVL C01996 V=800.0 PL=0
MOVL C01997 V=800.0 PL=0
MOVL C01998 V=800.0 PL=0
MOVL C01999 V=800.0 PL=0
MOVL C02000 V=800.0 PL=0
MOVL C02001 V=800.0 PL=0
MOVL C02002 V=800.0 PL=0
MOVL C02003 V=800.0 PL=0
MOVL C02004 V=800.0 PL=0
MOVL C02005 V=800.0 PL=0
MOVL C02006 V=800.0 PL=0
MOVL C02007 V=800.0 PL=0
MOVL C02008 V=800.0 PL=0
MOVL C02009 V=800.0 PL=0
MOVL C02010 V=800.0 PL=0
MOVL C02011 V=800.0 PL=0
MOVL C02012 V=800.0 PL=0
MOVL C02013 V=800.0 PL=0
MOVL C02014 V=800.0 PL=0
MOVL C02015 V=800.0 PL=0
MOVL C02016 V=800.0 PL=0
MOVL C02017 V=800.0 PL=0
MOVL C02018 V=800.0 PL=0
MOVL C02019 V=800.0 PL=0
MOVL C02020 V=800.0 PL=0
MOVL C02021 V=800.0 PL=0
MOVL C02022 V=800.0 PL=0
MOVL C02023 V=800.0 PL=0
MOVL C02024 V=800.0 PL=0
MOVL C02025 V=800.0 PL=0
MOVL C02026 V=800.0 PL=0
MOVL C02027 V=800.0 PL=0
MOVL C02028 V=800.0 PL=0
MOVL C02029 V=800.0 PL=0
MOVL C02030 V=800.0 PL=0
MOVL C02031 V=800.0 PL=0
MOVL C02032 V=800.0 PL=0
MOVL C02033 V=800.0 PL=0
MOVL C02034 V=800.0 PL=0
MOVL C02035 V=800.0 PL=0
MOVL C02036 V=800.0 PL=0
MOVL C02037 V=800.0 PL=0
MOVL C02038 V=800.0 PL=0
MOVL C02039 V=800.0 PL=0
MOVL C02040 V=800.0 PL=0
MOVL C02041 V=800.0 PL=0
MOVL C02042 V=800.0 PL=0
MOVL C02043 V=800.0 PL=0
MOVL C02044 V=800.0 PL=0
MOVL C02045 V=800.0 PL=0
MOVL C02046 V=800.0 PL=0
MOVL C02047 V=800.0 PL=0
MOVL C02048 V=800.0 PL=0
MOVL C02049 V=800.0 PL=0
MOVL C02050 V=800.0 PL=0
MOVL C02051 V=800.0 PL=0
MOVL C02052 V=800.0 PL=0
MOVL C02053 V=800.0 PL=0
MOVL C02054 V=800.0 PL=0
MOVL C02055 V=800.0 PL=0
MOVL C02056 V=800.0 PL=0
MOVL C02057 V=800.0 PL=0
MOVL C02058 V=800.0 PL=0
MOVL C02059 V=800.0 PL=0
MOVL C02060 V=800.0 PL=0
MOVL C02061 V=800.0 PL=0
MOVL C02062 V=800.0 PL=0
MOVL C02063 V=800.0 PL=0
MOVL C02064 V=800.0 PL=0
MOVL C02065 V=800.0 PL=0
MOVL C02066 V=800.0 PL=0
MOVL C02067 V=800.0 PL=0
MOVL C02068 V=800.0 PL=0
MOVL C02069 V=800.0 PL=0
MOVL C02070 V=800.0 PL=0
MOVL C02071 V=800.0 PL=0
MOVL C02072 V=800.0 PL=0
MOVL C02073 V=800.0 PL=0
MOVL C02074 V=800.0 PL=0
MOVL C02075 V=800.0 PL=0
MOVL C02076 V=800.0 PL=0
MOVL C02077 V=800.0 PL=0
MOVL C02078 V=800.0 PL=0
MOVL C02079 V=800.0 PL=0
MOVL C02080 V=800.0 PL=0
MOVL C02081 V=800.0 PL=0
MOVL C02082 V=800.0 PL=0
MOVL C02083 V=800.0 PL=0
MOVL C02084 V=800.0 PL=0
MOVL C02085 V=800.0 PL=0
MOVL C02086 V=800.0 PL=0
MOVL C02087 V=800.0 PL=0
MOVL C02088 V=800.0 PL=0
MOVL C02089 V=800.0 PL=0
MOVL C02090 V=800.0 PL=0
MOVL C02091 V=800.0 PL=0
MOVL C02092 V=800.0 PL=0
MOVL C02093 V=800.0 PL=0
MOVL C02094 V=800.0 PL=0
MOVL C02095 V=800.0 PL=0
MOVL C02096 V=800.0 PL=0
MOVL C02097 V=800.0 PL=0
MOVL C02098 V=800.0 PL=0
MOVL C02099 V=800.0 PL=0
MOVL C02100 V=800.0 PL=0
MOVL C02101 V=800.0 PL=0
MOVL C02102 V=800.0 PL=0
MOVL C02103 V=800.0 PL=0
MOVL C02104 V=800.0 PL=0
MOVL C02105 V=800.0 PL=0
MOVL C02106 V=800.0 PL=0
MOVL C02107 V=800.0 PL=0
MOVL C02108 V=800.0 PL=0
MOVL C02109 V=800.0 PL=0
MOVL C02110 V=800.0 PL=0
MOVL C02111 V=800.0 PL=0
MOVL C02112 V=800.0 PL=0
MOVL C02113 V=800.0 PL=0
MOVL C02114 V=800.0 PL=0
MOVL C02115 V=800.0 PL=0
MOVL C02116 V=800.0 PL=0
MOVL C02117 V=800.0 PL=0
MOVL C02118 V=800.0 PL=0
MOVL C02119 V=800.0 PL=0
MOVL C02120 V=800.0 PL=0
MOVL C02121 V=800.0 PL=0
MOVL C02122 V=800.0 PL=0
MOVL C02123 V=800.0 PL=0
MOVL C02124 V=800.0 PL=0
MOVL C02125 V=800.0 PL=0
MOVL C02126 V=800.0 PL=0
MOVL C02127 V=800.0 PL=0
MOVL C02128 V=800.0 PL=0
MOVL C02129 V=800.0 PL=0
MOVL C02130 V=800.0 PL=0
MOVL C02131 V=800.0 PL=0
MOVL C02132 V=800.0 PL=0
MOVL C02133 V=800.0 PL=0
MOVL C02134 V=800.0 PL=0
MOVL C02135 V=800.0 PL=0
MOVL C02136 V=800.0 PL=0
MOVL C02137 V=800.0 PL=0
MOVL C02138 V=800.0 PL=0
MOVL C02139 V=800.0 PL=0
MOVL C02140 V=800.0 PL=0
MOVL C02141 V=800.0 PL=0
MOVL C02142 V=800.0 PL=0
MOVL C02143 V=800.0 PL=0
MOVL C02144 V=800.0 PL=0
MOVL C02145 V=800.0 PL=0
MOVL C02146 V=800.0 PL=0
MOVL C02147 V=800.0 PL=0
MOVL C02148 V=800.0 PL=0
MOVL C02149 V=800.0 PL=0
MOVL C02150 V=800.0 PL=0
MOVL C02151 V=800.0 PL=0
MOVL C02152 V=800.0 PL=0
MOVL C02153 V=800.0 PL=0
MOVL C02154 V=800.0 PL=0
MOVL C02155 V=800.0 PL=0
